	VAR robtarget Openhole_1385 := [[446.82, -4.21, 181.42], [-0.057245, 0.704786, 0.705942, -0.040573], [0,0,0,0], [9E9, 9E9, 9E9, 9E9, 9E9, 9E9]];
	VAR robtarget Openhole_1386 := [[447.31, -4.15, 181.35], [-0.055802, 0.704902, 0.705831, -0.042464], [0,0,0,0], [9E9, 9E9, 9E9, 9E9, 9E9, 9E9]];
	VAR robtarget Openhole_1387 := [[447.8, -4.1, 181.28], [-0.0543, 0.705019, 0.705717, -0.044309], [0,0,0,0], [9E9, 9E9, 9E9, 9E9, 9E9, 9E9]];
	VAR robtarget Openhole_1388 := [[448.3, -4.06, 181.21], [-0.052766, 0.705135, 0.705601, -0.046125], [0,0,0,0], [9E9, 9E9, 9E9, 9E9, 9E9, 9E9]];
	VAR robtarget Openhole_1389 := [[448.79, -4.06, 181.14], [-0.051091, 0.705259, 0.705489, -0.047811], [0,0,0,0], [9E9, 9E9, 9E9, 9E9, 9E9, 9E9]];
	VAR robtarget Openhole_1390 := [[449.78, -4.1, 181], [-0.047615, 0.705502, 0.705261, -0.051054], [0,0,0,0], [9E9, 9E9, 9E9, 9E9, 9E9, 9E9]];
	VAR robtarget Openhole_1391 := [[450.77, -4.2, 180.86], [-0.043933, 0.705741, 0.705037, -0.05406], [0,0,0,0], [9E9, 9E9, 9E9, 9E9, 9E9, 9E9]];
	VAR robtarget Openhole_1392 := [[456.16, -5.01, 180.14], [-0.022875, 0.706737, 0.703678, -0.069553], [0,0,0,0], [9E9, 9E9, 9E9, 9E9, 9E9, 9E9]];
	VAR robtarget Openhole_1393 := [[458.63, -5.19, 179.82], [-0.013826, 0.706972, 0.702881, -0.077186], [0,0,0,0], [9E9, 9E9, 9E9, 9E9, 9E9, 9E9]];
	VAR robtarget Openhole_1394 := [[459.13, -5.2, 179.76], [-0.012101, 0.707003, 0.702703, -0.078798], [0,0,0,0], [9E9, 9E9, 9E9, 9E9, 9E9, 9E9]];
	VAR robtarget Openhole_1395 := [[463.08, -5.04, 179.21], [0.000809, 0.707106, 0.701046, -0.092383], [0,0,0,0], [9E9, 9E9, 9E9, 9E9, 9E9, 9E9]];
	VAR robtarget Openhole_1396 := [[464.07, -4.96, 179.07], [0.003883, 0.707096, 0.700578, -0.095868], [0,0,0,0], [9E9, 9E9, 9E9, 9E9, 9E9, 9E9]];
	VAR robtarget Openhole_1397 := [[472.91, -4.06, 177.66], [0.03065, 0.706442, 0.695628, -0.126894], [0,0,0,0], [9E9, 9E9, 9E9, 9E9, 9E9, 9E9]];
	VAR robtarget Openhole_1398 := [[478.34, -3.86, 176.83], [0.047884, 0.705484, 0.69228, -0.144041], [0,0,0,0], [9E9, 9E9, 9E9, 9E9, 9E9, 9E9]];
	VAR robtarget Openhole_1399 := [[478.84, -3.85, 176.75], [0.049491, 0.705373, 0.691972, -0.145517], [0,0,0,0], [9E9, 9E9, 9E9, 9E9, 9E9, 9E9]];
	VAR robtarget Openhole_1400 := [[479.33, -3.86, 176.68], [0.051109, 0.705257, 0.691664, -0.146975], [0,0,0,0], [9E9, 9E9, 9E9, 9E9, 9E9, 9E9]];
	VAR robtarget Openhole_1401 := [[480.82, -3.88, 176.47], [0.055996, 0.704886, 0.690737, -0.151267], [0,0,0,0], [9E9, 9E9, 9E9, 9E9, 9E9, 9E9]];
	VAR robtarget Openhole_1402 := [[474.12, -5.49, 177.83], [0.039301, 0.706014, 0.69579, -0.126003], [0,0,0,0], [9E9, 9E9, 9E9, 9E9, 9E9, 9E9]];
	VAR robtarget Openhole_1403 := [[469.2, -6.03, 178.58], [0.024725, 0.706674, 0.698676, -0.108864], [0,0,0,0], [9E9, 9E9, 9E9, 9E9, 9E9, 9E9]];
	VAR robtarget Openhole_1404 := [[460.88, -7.27, 179.76], [0.000748, 0.707106, 0.702821, -0.077733], [0,0,0,0], [9E9, 9E9, 9E9, 9E9, 9E9, 9E9]];
	VAR robtarget Openhole_1405 := [[457.42, -7.57, 180.17], [-0.010045, 0.707035, 0.704092, -0.065225], [0,0,0,0], [9E9, 9E9, 9E9, 9E9, 9E9, 9E9]];
	VAR robtarget Openhole_1406 := [[455.43, -7.61, 180.39], [-0.016666, 0.70691, 0.70469, -0.058409], [0,0,0,0], [9E9, 9E9, 9E9, 9E9, 9E9, 9E9]];
	VAR robtarget Openhole_1407 := [[452.45, -7.48, 180.72], [-0.027253, 0.706581, 0.705422, -0.048789], [0,0,0,0], [9E9, 9E9, 9E9, 9E9, 9E9, 9E9]];
	VAR robtarget Openhole_1408 := [[448.48, -7.26, 181.16], [-0.041479, 0.705889, 0.706188, -0.036043], [0,0,0,0], [9E9, 9E9, 9E9, 9E9, 9E9, 9E9]];
	VAR robtarget Openhole_1409 := [[447.49, -7.25, 181.27], [-0.044879, 0.705681, 0.706351, -0.032691], [0,0,0,0], [9E9, 9E9, 9E9, 9E9, 9E9, 9E9]];
	VAR robtarget Openhole_1410 := [[446.49, -7.27, 181.38], [-0.048173, 0.705464, 0.706502, -0.029233], [0,0,0,0], [9E9, 9E9, 9E9, 9E9, 9E9, 9E9]];
	VAR robtarget Openhole_1411 := [[445.5, -7.33, 181.49], [-0.051296, 0.705244, 0.706642, -0.025622], [0,0,0,0], [9E9, 9E9, 9E9, 9E9, 9E9, 9E9]];
	VAR robtarget Openhole_1412 := [[444.51, -7.43, 181.6], [-0.054297, 0.705019, 0.706767, -0.021908], [0,0,0,0], [9E9, 9E9, 9E9, 9E9, 9E9, 9E9]];
	VAR robtarget Openhole_1413 := [[444.02, -7.49, 181.65], [-0.055764, 0.704905, 0.706823, -0.020026], [0,0,0,0], [9E9, 9E9, 9E9, 9E9, 9E9, 9E9]];
	VAR robtarget Openhole_1414 := [[437.6, -8.31, 182.27], [-0.074416, 0.70318, 0.707092, 0.004635], [0,0,0,0], [9E9, 9E9, 9E9, 9E9, 9E9, 9E9]];
	VAR robtarget Openhole_1415 := [[423.69, -9.33, 183.46], [-0.115694, 0.697578, 0.704998, 0.05457], [0,0,0,0], [9E9, 9E9, 9E9, 9E9, 9E9, 9E9]];
	VAR robtarget Openhole_1416 := [[407.25, -10.08, 184.69], [-0.161587, 0.688396, 0.698742, 0.108443], [0,0,0,0], [9E9, 9E9, 9E9, 9E9, 9E9, 9E9]];
	VAR robtarget Openhole_1417 := [[394.36, -10.64, 185.5], [-0.193652, 0.680073, 0.691718, 0.14672], [0,0,0,0], [9E9, 9E9, 9E9, 9E9, 9E9, 9E9]];
	VAR robtarget Openhole_1418 := [[389.36, -10.64, 185.9], [-0.205704, 0.676525, 0.688791, 0.159896], [0,0,0,0], [9E9, 9E9, 9E9, 9E9, 9E9, 9E9]];
	VAR robtarget Openhole_1419 := [[362.36, -10.64, 185.99], [-0.183051, 0.683002, 0.683002, 0.183051], [0,0,0,0], [9E9, 9E9, 9E9, 9E9, 9E9, 9E9]];
	VAR robtarget Openhole_1420 := [[361.72, -33.92, 172.54], [-0.183051, 0.683002, 0.683002, 0.183051], [0,0,0,0], [9E9, 9E9, 9E9, 9E9, 9E9, 9E9]];
	VAR robtarget Openhole_1421 := [[389.32, -33.92, 172.46], [-0.13956, 0.693198, 0.67011, 0.225726], [0,0,0,0], [9E9, 9E9, 9E9, 9E9, 9E9, 9E9]];
	VAR robtarget Openhole_1422 := [[399.12, -33.92, 173.86], [-0.112191, 0.69815, 0.677451, 0.202632], [0,0,0,0], [9E9, 9E9, 9E9, 9E9, 9E9, 9E9]];
	VAR robtarget Openhole_1423 := [[405.5, -35.06, 174.3], [-0.089819, 0.701379, 0.681181, 0.189715], [0,0,0,0], [9E9, 9E9, 9E9, 9E9, 9E9, 9E9]];
	VAR robtarget Openhole_1424 := [[411.91, -35.92, 174.98], [-0.067308, 0.703896, 0.685089, 0.175081], [0,0,0,0], [9E9, 9E9, 9E9, 9E9, 9E9, 9E9]];
	VAR robtarget Openhole_1425 := [[417.83, -36.39, 175.8], [-0.046793, 0.705557, 0.688811, 0.159812], [0,0,0,0], [9E9, 9E9, 9E9, 9E9, 9E9, 9E9]];
	VAR robtarget Openhole_1426 := [[421.78, -36.5, 176.43], [-0.033466, 0.706314, 0.691318, 0.148591], [0,0,0,0], [9E9, 9E9, 9E9, 9E9, 9E9, 9E9]];
	VAR robtarget Openhole_1427 := [[422.28, -36.5, 176.51], [-0.031833, 0.70639, 0.691632, 0.147122], [0,0,0,0], [9E9, 9E9, 9E9, 9E9, 9E9, 9E9]];
	VAR robtarget Openhole_1428 := [[428.18, -36.31, 177.54], [-0.012705, 0.706993, 0.695332, 0.128505], [0,0,0,0], [9E9, 9E9, 9E9, 9E9, 9E9, 9E9]];
	VAR robtarget Openhole_1429 := [[436.05, -35.81, 178.91], [0.012379, 0.706998, 0.699726, 0.101898], [0,0,0,0], [9E9, 9E9, 9E9, 9E9, 9E9, 9E9]];
	VAR robtarget Openhole_1430 := [[437.03, -35.79, 179.08], [0.015677, 0.706933, 0.700196, 0.098619], [0,0,0,0], [9E9, 9E9, 9E9, 9E9, 9E9, 9E9]];
	VAR robtarget Openhole_1431 := [[438.02, -35.8, 179.23], [0.019061, 0.70685, 0.700641, 0.095405], [0,0,0,0], [9E9, 9E9, 9E9, 9E9, 9E9, 9E9]];
	VAR robtarget Openhole_1432 := [[439.01, -35.82, 179.39], [0.022528, 0.706748, 0.701062, 0.092258], [0,0,0,0], [9E9, 9E9, 9E9, 9E9, 9E9, 9E9]];
	VAR robtarget Openhole_1433 := [[439.99, -35.88, 179.55], [0.026095, 0.706625, 0.701458, 0.089204], [0,0,0,0], [9E9, 9E9, 9E9, 9E9, 9E9, 9E9]];
	VAR robtarget Openhole_1434 := [[440.98, -35.98, 179.7], [0.029757, 0.70648, 0.701827, 0.086247], [0,0,0,0], [9E9, 9E9, 9E9, 9E9, 9E9, 9E9]];
	VAR robtarget Openhole_1435 := [[441.96, -36.1, 179.85], [0.03352, 0.706312, 0.702171, 0.083404], [0,0,0,0], [9E9, 9E9, 9E9, 9E9, 9E9, 9E9]];
	VAR robtarget Openhole_1436 := [[442.94, -36.26, 180], [0.037368, 0.706119, 0.702491, 0.080666], [0,0,0,0], [9E9, 9E9, 9E9, 9E9, 9E9, 9E9]];
	VAR robtarget Openhole_1437 := [[443.91, -36.44, 180.15], [0.041287, 0.7059, 0.702789, 0.078026], [0,0,0,0], [9E9, 9E9, 9E9, 9E9, 9E9, 9E9]];
	VAR robtarget Openhole_1438 := [[445.84, -36.87, 180.46], [0.049255, 0.705389, 0.703335, 0.072942], [0,0,0,0], [9E9, 9E9, 9E9, 9E9, 9E9, 9E9]];
	VAR robtarget Openhole_1439 := [[446.31, -37, 180.54], [0.051325, 0.705242, 0.703452, 0.071803], [0,0,0,0], [9E9, 9E9, 9E9, 9E9, 9E9, 9E9]];
	VAR robtarget Openhole_1440 := [[446.78, -37.17, 180.61], [0.05345, 0.705084, 0.703556, 0.070775], [0,0,0,0], [9E9, 9E9, 9E9, 9E9, 9E9, 9E9]];
	VAR robtarget Openhole_1441 := [[447.23, -37.35, 180.69], [0.05561, 0.704917, 0.70365, 0.06983], [0,0,0,0], [9E9, 9E9, 9E9, 9E9, 9E9, 9E9]];
	VAR robtarget Openhole_1442 := [[448.2, -37.57, 180.86], [0.059582, 0.704592, 0.703898, 0.067287], [0,0,0,0], [9E9, 9E9, 9E9, 9E9, 9E9, 9E9]];
	VAR robtarget Openhole_1443 := [[448.69, -37.57, 180.94], [0.061268, 0.704447, 0.704054, 0.06564], [0,0,0,0], [9E9, 9E9, 9E9, 9E9, 9E9, 9E9]];
	VAR robtarget Openhole_1444 := [[449.18, -37.57, 181.03], [0.06291, 0.704303, 0.704209, 0.063947], [0,0,0,0], [9E9, 9E9, 9E9, 9E9, 9E9, 9E9]];
	VAR robtarget Openhole_1445 := [[450.15, -37.36, 181.2], [0.065502, 0.704066, 0.704556, 0.060003], [0,0,0,0], [9E9, 9E9, 9E9, 9E9, 9E9, 9E9]];
	VAR robtarget Openhole_1446 := [[450.62, -37.23, 181.28], [0.066679, 0.703956, 0.704728, 0.057956], [0,0,0,0], [9E9, 9E9, 9E9, 9E9, 9E9, 9E9]];
	VAR robtarget Openhole_1447 := [[451.1, -37.12, 181.37], [0.067916, 0.703838, 0.70489, 0.055943], [0,0,0,0], [9E9, 9E9, 9E9, 9E9, 9E9, 9E9]];
	VAR robtarget Openhole_1448 := [[451.58, -36.98, 181.45], [0.069072, 0.703725, 0.705051, 0.053881], [0,0,0,0], [9E9, 9E9, 9E9, 9E9, 9E9, 9E9]];
	VAR robtarget Openhole_1449 := [[459.65, -34.59, 182.6], [0.088061, 0.701602, 0.706869, 0.01833], [0,0,0,0], [9E9, 9E9, 9E9, 9E9, 9E9, 9E9]];
	VAR robtarget Openhole_1450 := [[460.13, -34.45, 182.66], [0.089197, 0.701458, 0.70692, 0.01625], [0,0,0,0], [9E9, 9E9, 9E9, 9E9, 9E9, 9E9]];
	VAR robtarget Openhole_1451 := [[461.11, -32.96, 182.64], [0.087508, 0.701671, 0.707062, 0.00793], [0,0,0,0], [9E9, 9E9, 9E9, 9E9, 9E9, 9E9]];
	VAR robtarget Openhole_1452 := [[460.14, -33.18, 182.53], [0.085056, 0.701973, 0.707005, 0.01198], [0,0,0,0], [9E9, 9E9, 9E9, 9E9, 9E9, 9E9]];
	VAR robtarget Openhole_1453 := [[453.43, -34.99, 181.69], [0.068762, 0.703755, 0.705919, 0.040973], [0,0,0,0], [9E9, 9E9, 9E9, 9E9, 9E9, 9E9]];
	VAR robtarget Openhole_1454 := [[452.47, -35.23, 181.55], [0.066291, 0.703993, 0.705672, 0.045027], [0,0,0,0], [9E9, 9E9, 9E9, 9E9, 9E9, 9E9]];
	VAR robtarget Openhole_1455 := [[451.98, -35.33, 181.48], [0.065007, 0.704112, 0.705542, 0.047022], [0,0,0,0], [9E9, 9E9, 9E9, 9E9, 9E9, 9E9]];
	VAR robtarget Openhole_1456 := [[451.5, -35.42, 181.4], [0.063682, 0.704233, 0.705408, 0.048988], [0,0,0,0], [9E9, 9E9, 9E9, 9E9, 9E9, 9E9]];
	VAR robtarget Openhole_1457 := [[451.01, -35.49, 181.32], [0.062259, 0.704361, 0.705274, 0.050884], [0,0,0,0], [9E9, 9E9, 9E9, 9E9, 9E9, 9E9]];
	VAR robtarget Openhole_1458 := [[450.52, -35.55, 181.25], [0.06079, 0.704489, 0.705137, 0.052742], [0,0,0,0], [9E9, 9E9, 9E9, 9E9, 9E9, 9E9]];
	VAR robtarget Openhole_1459 := [[450.03, -35.58, 181.17], [0.059241, 0.704621, 0.705001, 0.054535], [0,0,0,0], [9E9, 9E9, 9E9, 9E9, 9E9, 9E9]];
	VAR robtarget Openhole_1460 := [[449.53, -35.6, 181.09], [0.057631, 0.704754, 0.704864, 0.056273], [0,0,0,0], [9E9, 9E9, 9E9, 9E9, 9E9, 9E9]];
	VAR robtarget Openhole_1461 := [[449.04, -35.59, 181.01], [0.055918, 0.704892, 0.704732, 0.057906], [0,0,0,0], [9E9, 9E9, 9E9, 9E9, 9E9, 9E9]];
	VAR robtarget Openhole_1462 := [[448.55, -35.55, 180.93], [0.054128, 0.705032, 0.704603, 0.059455], [0,0,0,0], [9E9, 9E9, 9E9, 9E9, 9E9, 9E9]];
	VAR robtarget Openhole_1463 := [[448.05, -35.5, 180.86], [0.052284, 0.705171, 0.704476, 0.060939], [0,0,0,0], [9E9, 9E9, 9E9, 9E9, 9E9, 9E9]];
	VAR robtarget Openhole_1464 := [[447.57, -35.43, 180.78], [0.050389, 0.705309, 0.704352, 0.062358], [0,0,0,0], [9E9, 9E9, 9E9, 9E9, 9E9, 9E9]];
	VAR robtarget Openhole_1465 := [[446.59, -35.25, 180.63], [0.046491, 0.705577, 0.704108, 0.065048], [0,0,0,0], [9E9, 9E9, 9E9, 9E9, 9E9, 9E9]];
	VAR robtarget Openhole_1466 := [[443.68, -34.65, 180.21], [0.034621, 0.706259, 0.703341, 0.072881], [0,0,0,0], [9E9, 9E9, 9E9, 9E9, 9E9, 9E9]];
	VAR robtarget Openhole_1467 := [[441.72, -34.35, 179.94], [0.026944, 0.706593, 0.702744, 0.078425], [0,0,0,0], [9E9, 9E9, 9E9, 9E9, 9E9, 9E9]];
	VAR robtarget Openhole_1468 := [[440.74, -34.25, 179.8], [0.023237, 0.706725, 0.702411, 0.081357], [0,0,0,0], [9E9, 9E9, 9E9, 9E9, 9E9, 9E9]];
	VAR robtarget Openhole_1469 := [[439.75, -34.17, 179.66], [0.019621, 0.706835, 0.702053, 0.084386], [0,0,0,0], [9E9, 9E9, 9E9, 9E9, 9E9, 9E9]];
	VAR robtarget Openhole_1470 := [[438.76, -34.13, 179.52], [0.016102, 0.706923, 0.701671, 0.087509], [0,0,0,0], [9E9, 9E9, 9E9, 9E9, 9E9, 9E9]];
	VAR robtarget Openhole_1471 := [[437.77, -34.12, 179.38], [0.012688, 0.706993, 0.701262, 0.090726], [0,0,0,0], [9E9, 9E9, 9E9, 9E9, 9E9, 9E9]];
	VAR robtarget Openhole_1472 := [[437.28, -34.12, 179.31], [0.011017, 0.707021, 0.701049, 0.092362], [0,0,0,0], [9E9, 9E9, 9E9, 9E9, 9E9, 9E9]];
	VAR robtarget Openhole_1473 := [[431.85, -34.44, 178.47], [-0.006368, 0.707078, 0.698349, 0.110947], [0,0,0,0], [9E9, 9E9, 9E9, 9E9, 9E9, 9E9]];
	VAR robtarget Openhole_1474 := [[424.96, -34.89, 177.34], [-0.028091, 0.706549, 0.694309, 0.13392], [0,0,0,0], [9E9, 9E9, 9E9, 9E9, 9E9, 9E9]];
	VAR robtarget Openhole_1475 := [[422, -34.94, 176.87], [-0.037745, 0.706099, 0.692485, 0.143054], [0,0,0,0], [9E9, 9E9, 9E9, 9E9, 9E9, 9E9]];
	VAR robtarget Openhole_1476 := [[421.5, -34.94, 176.8], [-0.039386, 0.706009, 0.69218, 0.144521], [0,0,0,0], [9E9, 9E9, 9E9, 9E9, 9E9, 9E9]];
	VAR robtarget Openhole_1477 := [[415.57, -34.71, 175.97], [-0.059446, 0.704604, 0.688505, 0.161124], [0,0,0,0], [9E9, 9E9, 9E9, 9E9, 9E9, 9E9]];
	VAR robtarget Openhole_1478 := [[409.14, -34.09, 175.23], [-0.08164, 0.702378, 0.684557, 0.177147], [0,0,0,0], [9E9, 9E9, 9E9, 9E9, 9E9, 9E9]];
	VAR robtarget Openhole_1479 := [[404.2, -33.45, 174.8], [-0.098663, 0.70019, 0.681563, 0.18834], [0,0,0,0], [9E9, 9E9, 9E9, 9E9, 9E9, 9E9]];
	VAR robtarget Openhole_1480 := [[411.67, -32.92, 176.03], [-0.077413, 0.702856, 0.687197, 0.166612], [0,0,0,0], [9E9, 9E9, 9E9, 9E9, 9E9, 9E9]];
	VAR robtarget Openhole_1481 := [[418.12, -33.28, 176.78], [-0.055758, 0.704905, 0.691162, 0.149313], [0,0,0,0], [9E9, 9E9, 9E9, 9E9, 9E9, 9E9]];
	VAR robtarget Openhole_1482 := [[420.59, -33.32, 177.11], [-0.047583, 0.705504, 0.69268, 0.142107], [0,0,0,0], [9E9, 9E9, 9E9, 9E9, 9E9, 9E9]];
	VAR robtarget Openhole_1483 := [[421.09, -33.31, 177.18], [-0.04597, 0.705611, 0.692983, 0.14062], [0,0,0,0], [9E9, 9E9, 9E9, 9E9, 9E9, 9E9]];
	VAR robtarget Openhole_1484 := [[426.52, -33.08, 177.98], [-0.028736, 0.706523, 0.696271, 0.123317], [0,0,0,0], [9E9, 9E9, 9E9, 9E9, 9E9, 9E9]];
	VAR robtarget Openhole_1485 := [[436.37, -32.09, 179.43], [0.001182, 0.707106, 0.701528, 0.088645], [0,0,0,0], [9E9, 9E9, 9E9, 9E9, 9E9, 9E9]];
	VAR robtarget Openhole_1486 := [[438.84, -31.99, 179.75], [0.009265, 0.707046, 0.702549, 0.080151], [0,0,0,0], [9E9, 9E9, 9E9, 9E9, 9E9, 9E9]];
	VAR robtarget Openhole_1487 := [[439.84, -31.99, 179.88], [0.012667, 0.706993, 0.702914, 0.076885], [0,0,0,0], [9E9, 9E9, 9E9, 9E9, 9E9, 9E9]];
	VAR robtarget Openhole_1488 := [[441.32, -32.04, 180.06], [0.017908, 0.70688, 0.703421, 0.072104], [0,0,0,0], [9E9, 9E9, 9E9, 9E9, 9E9, 9E9]];
	VAR robtarget Openhole_1489 := [[442.32, -32.11, 180.18], [0.0215, 0.70678, 0.703731, 0.069008], [0,0,0,0], [9E9, 9E9, 9E9, 9E9, 9E9, 9E9]];
	VAR robtarget Openhole_1490 := [[442.81, -32.16, 180.24], [0.023347, 0.706721, 0.703876, 0.067516], [0,0,0,0], [9E9, 9E9, 9E9, 9E9, 9E9, 9E9]];
	VAR robtarget Openhole_1491 := [[447.23, -32.82, 180.78], [0.040592, 0.705941, 0.704977, 0.054843], [0,0,0,0], [9E9, 9E9, 9E9, 9E9, 9E9, 9E9]];
	VAR robtarget Openhole_1492 := [[448.21, -32.96, 180.91], [0.044393, 0.705712, 0.705193, 0.051985], [0,0,0,0], [9E9, 9E9, 9E9, 9E9, 9E9, 9E9]];
	VAR robtarget Openhole_1493 := [[448.7, -33.01, 180.97], [0.046239, 0.705593, 0.705302, 0.050486], [0,0,0,0], [9E9, 9E9, 9E9, 9E9, 9E9, 9E9]];
	VAR robtarget Openhole_1494 := [[449.19, -33.05, 181.04], [0.048038, 0.705473, 0.705412, 0.048933], [0,0,0,0], [9E9, 9E9, 9E9, 9E9, 9E9, 9E9]];
	VAR robtarget Openhole_1495 := [[449.69, -33.07, 181.11], [0.049788, 0.705352, 0.705521, 0.047323], [0,0,0,0], [9E9, 9E9, 9E9, 9E9, 9E9, 9E9]];
	VAR robtarget Openhole_1496 := [[450.19, -33.08, 181.17], [0.051486, 0.70523, 0.705631, 0.045656], [0,0,0,0], [9E9, 9E9, 9E9, 9E9, 9E9, 9E9]];
	VAR robtarget Openhole_1497 := [[451.18, -33.03, 181.31], [0.054685, 0.704989, 0.70585, 0.042136], [0,0,0,0], [9E9, 9E9, 9E9, 9E9, 9E9, 9E9]];
	VAR robtarget Openhole_1498 := [[451.67, -32.99, 181.37], [0.056197, 0.70487, 0.705957, 0.0403], [0,0,0,0], [9E9, 9E9, 9E9, 9E9, 9E9, 9E9]];
	VAR robtarget Openhole_1499 := [[452.16, -32.92, 181.44], [0.057637, 0.704754, 0.706063, 0.038404], [0,0,0,0], [9E9, 9E9, 9E9, 9E9, 9E9, 9E9]];
	VAR robtarget Openhole_1500 := [[452.65, -32.84, 181.5], [0.059027, 0.704639, 0.706166, 0.036472], [0,0,0,0], [9E9, 9E9, 9E9, 9E9, 9E9, 9E9]];
	VAR robtarget Openhole_1501 := [[453.62, -32.66, 181.62], [0.061679, 0.704412, 0.706359, 0.032514], [0,0,0,0], [9E9, 9E9, 9E9, 9E9, 9E9, 9E9]];
	VAR robtarget Openhole_1502 := [[460.43, -31.22, 182.36], [0.079553, 0.702618, 0.707093, 0.004412], [0,0,0,0], [9E9, 9E9, 9E9, 9E9, 9E9, 9E9]];
	VAR robtarget Openhole_1503 := [[466.84, -30.31, 182.96], [0.097392, 0.700368, 0.706813, -0.020389], [0,0,0,0], [9E9, 9E9, 9E9, 9E9, 9E9, 9E9]];
	VAR robtarget Openhole_1504 := [[476.26, -29.36, 183.74], [0.123815, 0.696182, 0.704976, -0.054856], [0,0,0,0], [9E9, 9E9, 9E9, 9E9, 9E9, 9E9]];
	VAR robtarget Openhole_1505 := [[470.3, -26.56, 182.58], [0.096146, 0.70054, 0.70571, -0.044425], [0,0,0,0], [9E9, 9E9, 9E9, 9E9, 9E9, 9E9]];
	VAR robtarget Openhole_1506 := [[465.31, -26.64, 182.23], [0.080362, 0.702525, 0.706573, -0.027466], [0,0,0,0], [9E9, 9E9, 9E9, 9E9, 9E9, 9E9]];
	VAR robtarget Openhole_1507 := [[464.81, -26.64, 182.19], [0.078734, 0.70271, 0.706636, -0.02579], [0,0,0,0], [9E9, 9E9, 9E9, 9E9, 9E9, 9E9]];
	VAR robtarget Openhole_1508 := [[463.82, -26.63, 182.12], [0.075461, 0.703069, 0.706751, -0.022436], [0,0,0,0], [9E9, 9E9, 9E9, 9E9, 9E9, 9E9]];
	VAR robtarget Openhole_1509 := [[463.32, -26.64, 182.08], [0.07383, 0.703242, 0.706802, -0.020747], [0,0,0,0], [9E9, 9E9, 9E9, 9E9, 9E9, 9E9]];
	VAR robtarget Openhole_1510 := [[462.82, -26.63, 182.05], [0.072175, 0.703414, 0.706849, -0.019077], [0,0,0,0], [9E9, 9E9, 9E9, 9E9, 9E9, 9E9]];
	VAR robtarget Openhole_1511 := [[459.33, -26.59, 181.79], [0.060506, 0.704513, 0.707069, -0.007354], [0,0,0,0], [9E9, 9E9, 9E9, 9E9, 9E9, 9E9]];
	VAR robtarget Openhole_1512 := [[458.83, -26.59, 181.75], [0.058846, 0.704654, 0.707084, -0.005656], [0,0,0,0], [9E9, 9E9, 9E9, 9E9, 9E9, 9E9]];
	VAR robtarget Openhole_1513 := [[458.33, -26.6, 181.72], [0.057195, 0.70479, 0.707096, -0.003946], [0,0,0,0], [9E9, 9E9, 9E9, 9E9, 9E9, 9E9]];
	VAR robtarget Openhole_1514 := [[457.83, -26.59, 181.68], [0.055521, 0.704924, 0.707103, -0.002257], [0,0,0,0], [9E9, 9E9, 9E9, 9E9, 9E9, 9E9]];
	VAR robtarget Openhole_1515 := [[456.34, -26.58, 181.57], [0.050456, 0.705304, 0.707101, 0.002786], [0,0,0,0], [9E9, 9E9, 9E9, 9E9, 9E9, 9E9]];
	VAR robtarget Openhole_1516 := [[455.34, -26.54, 181.49], [0.046991, 0.705544, 0.707081, 0.006067], [0,0,0,0], [9E9, 9E9, 9E9, 9E9, 9E9, 9E9]];
	VAR robtarget Openhole_1517 := [[454.84, -26.49, 181.46], [0.045165, 0.705663, 0.707066, 0.007603], [0,0,0,0], [9E9, 9E9, 9E9, 9E9, 9E9, 9E9]];
	VAR robtarget Openhole_1518 := [[454.35, -26.44, 181.42], [0.043303, 0.70578, 0.707048, 0.009097], [0,0,0,0], [9E9, 9E9, 9E9, 9E9, 9E9, 9E9]];
	VAR robtarget Openhole_1519 := [[453.86, -26.35, 181.38], [0.041367, 0.705896, 0.707029, 0.010494], [0,0,0,0], [9E9, 9E9, 9E9, 9E9, 9E9, 9E9]];
	VAR robtarget Openhole_1520 := [[453.37, -26.25, 181.34], [0.039385, 0.706009, 0.707008, 0.011826], [0,0,0,0], [9E9, 9E9, 9E9, 9E9, 9E9, 9E9]];
	VAR robtarget Openhole_1521 := [[452.79, -25.92, 181.29], [0.0363, 0.706174, 0.706993, 0.012685], [0,0,0,0], [9E9, 9E9, 9E9, 9E9, 9E9, 9E9]];
	VAR robtarget Openhole_1522 := [[454.94, -24.42, 181.35], [0.038494, 0.706058, 0.707107, 0.000235], [0,0,0,0], [9E9, 9E9, 9E9, 9E9, 9E9, 9E9]];
	VAR robtarget Openhole_1523 := [[455.54, -24.57, 181.39], [0.041032, 0.705915, 0.707106, -0.001297], [0,0,0,0], [9E9, 9E9, 9E9, 9E9, 9E9, 9E9]];
	VAR robtarget Openhole_1524 := [[456.54, -24.66, 181.45], [0.044665, 0.705695, 0.707093, -0.004397], [0,0,0,0], [9E9, 9E9, 9E9, 9E9, 9E9, 9E9]];
	VAR robtarget Openhole_1525 := [[457.04, -24.68, 181.48], [0.046428, 0.705581, 0.707081, -0.006004], [0,0,0,0], [9E9, 9E9, 9E9, 9E9, 9E9, 9E9]];
	VAR robtarget Openhole_1526 := [[460.52, -24.98, 181.7], [0.059039, 0.704638, 0.706906, -0.016839], [0,0,0,0], [9E9, 9E9, 9E9, 9E9, 9E9, 9E9]];
	VAR robtarget Openhole_1527 := [[457.18, -28.45, 181.77], [0.059563, 0.704594, 0.707079, 0.006212], [0,0,0,0], [9E9, 9E9, 9E9, 9E9, 9E9, 9E9]];
	VAR robtarget Openhole_1528 := [[454.2, -28.65, 181.51], [0.050244, 0.705319, 0.706901, 0.017075], [0,0,0,0], [9E9, 9E9, 9E9, 9E9, 9E9, 9E9]];
	VAR robtarget Openhole_1529 := [[453.7, -28.66, 181.47], [0.048609, 0.705434, 0.706856, 0.018817], [0,0,0,0], [9E9, 9E9, 9E9, 9E9, 9E9, 9E9]];
	VAR robtarget Openhole_1530 := [[452.71, -28.67, 181.37], [0.045277, 0.705656, 0.706757, 0.022241], [0,0,0,0], [9E9, 9E9, 9E9, 9E9, 9E9, 9E9]];
	VAR robtarget Openhole_1531 := [[449.23, -28.52, 181.05], [0.033008, 0.706336, 0.706307, 0.033626], [0,0,0,0], [9E9, 9E9, 9E9, 9E9, 9E9, 9E9]];
	VAR robtarget Openhole_1532 := [[448.73, -28.52, 181.01], [0.031293, 0.706414, 0.706225, 0.035294], [0,0,0,0], [9E9, 9E9, 9E9, 9E9, 9E9, 9E9]];
	VAR robtarget Openhole_1533 := [[448.23, -28.52, 180.96], [0.029603, 0.706487, 0.706139, 0.036988], [0,0,0,0], [9E9, 9E9, 9E9, 9E9, 9E9, 9E9]];
	VAR robtarget Openhole_1534 := [[447.24, -28.52, 180.87], [0.02623, 0.70662, 0.705953, 0.040382], [0,0,0,0], [9E9, 9E9, 9E9, 9E9, 9E9, 9E9]];
	VAR robtarget Openhole_1535 := [[444.75, -28.61, 180.64], [0.018061, 0.706876, 0.7054, 0.049099], [0,0,0,0], [9E9, 9E9, 9E9, 9E9, 9E9, 9E9]];
	VAR robtarget Openhole_1536 := [[443.26, -28.67, 180.5], [0.013204, 0.706983, 0.705015, 0.054352], [0,0,0,0], [9E9, 9E9, 9E9, 9E9, 9E9, 9E9]];
	VAR robtarget Openhole_1537 := [[444.55, -31.6, 180.48], [0.027447, 0.706574, 0.704572, 0.059817], [0,0,0,0], [9E9, 9E9, 9E9, 9E9, 9E9, 9E9]];
	VAR robtarget Openhole_1538 := [[445.54, -31.73, 180.6], [0.03123, 0.706417, 0.704812, 0.056924], [0,0,0,0], [9E9, 9E9, 9E9, 9E9, 9E9, 9E9]];
	VAR robtarget Openhole_1539 := [[446.52, -31.9, 180.71], [0.035109, 0.706235, 0.70503, 0.05416], [0,0,0,0], [9E9, 9E9, 9E9, 9E9, 9E9, 9E9]];
	VAR robtarget Openhole_1540 := [[448.49, -32.14, 180.95], [0.042616, 0.705821, 0.705455, 0.048298], [0,0,0,0], [9E9, 9E9, 9E9, 9E9, 9E9, 9E9]];
	VAR robtarget Openhole_1541 := [[448.98, -32.18, 181.02], [0.044435, 0.705709, 0.705559, 0.046761], [0,0,0,0], [9E9, 9E9, 9E9, 9E9, 9E9, 9E9]];
	VAR robtarget Openhole_1542 := [[449.48, -32.21, 181.08], [0.046209, 0.705595, 0.705662, 0.045173], [0,0,0,0], [9E9, 9E9, 9E9, 9E9, 9E9, 9E9]];
	VAR robtarget Openhole_1543 := [[449.97, -32.23, 181.14], [0.047949, 0.705479, 0.705764, 0.043549], [0,0,0,0], [9E9, 9E9, 9E9, 9E9, 9E9, 9E9]];
	VAR robtarget Openhole_1544 := [[450.47, -32.23, 181.2], [0.049624, 0.705363, 0.705867, 0.041855], [0,0,0,0], [9E9, 9E9, 9E9, 9E9, 9E9, 9E9]];
	VAR robtarget Openhole_1545 := [[450.96, -32.22, 181.27], [0.051253, 0.705247, 0.705968, 0.04012], [0,0,0,0], [9E9, 9E9, 9E9, 9E9, 9E9, 9E9]];
	VAR robtarget Openhole_1546 := [[451.46, -32.18, 181.33], [0.052812, 0.705132, 0.706068, 0.038318], [0,0,0,0], [9E9, 9E9, 9E9, 9E9, 9E9, 9E9]];
	VAR robtarget Openhole_1547 := [[451.95, -32.13, 181.39], [0.05432, 0.705017, 0.706165, 0.036474], [0,0,0,0], [9E9, 9E9, 9E9, 9E9, 9E9, 9E9]];
	VAR robtarget Openhole_1548 := [[452.45, -32.07, 181.45], [0.055766, 0.704904, 0.706261, 0.03458], [0,0,0,0], [9E9, 9E9, 9E9, 9E9, 9E9, 9E9]];
	VAR robtarget Openhole_1549 := [[453.43, -31.9, 181.57], [0.058505, 0.704682, 0.706441, 0.030677], [0,0,0,0], [9E9, 9E9, 9E9, 9E9, 9E9, 9E9]];
	VAR robtarget Openhole_1550 := [[452.74, -30.49, 181.44], [0.051498, 0.705229, 0.706541, 0.028284], [0,0,0,0], [9E9, 9E9, 9E9, 9E9, 9E9, 9E9]];
	VAR robtarget Openhole_1551 := [[451.25, -30.57, 181.27], [0.046727, 0.705561, 0.706307, 0.033621], [0,0,0,0], [9E9, 9E9, 9E9, 9E9, 9E9, 9E9]];
	VAR robtarget Openhole_1552 := [[450.75, -30.57, 181.22], [0.045054, 0.70567, 0.706224, 0.035323], [0,0,0,0], [9E9, 9E9, 9E9, 9E9, 9E9, 9E9]];
	VAR robtarget Openhole_1553 := [[450.26, -30.57, 181.16], [0.043355, 0.705776, 0.706138, 0.036998], [0,0,0,0], [9E9, 9E9, 9E9, 9E9, 9E9, 9E9]];
	VAR robtarget Openhole_1554 := [[446.79, -30.31, 180.78], [0.030739, 0.706438, 0.70548, 0.047944], [0,0,0,0], [9E9, 9E9, 9E9, 9E9, 9E9, 9E9]];
	VAR robtarget Openhole_1555 := [[446.79, -30.31, 180.9], [0.030776, 0.706437, 0.705483, 0.047888], [0,0,0,0], [9E9, 9E9, 9E9, 9E9, 9E9, 9E9]];
	VAR robtarget Openhole_1556 := [[450.26, -30.57, 181.28], [0.043406, 0.705773, 0.70614, 0.036954], [0,0,0,0], [9E9, 9E9, 9E9, 9E9, 9E9, 9E9]];
	VAR robtarget Openhole_1557 := [[450.75, -30.57, 181.34], [0.045107, 0.705667, 0.706226, 0.035281], [0,0,0,0], [9E9, 9E9, 9E9, 9E9, 9E9, 9E9]];
	VAR robtarget Openhole_1558 := [[451.25, -30.57, 181.39], [0.046782, 0.705558, 0.706309, 0.033581], [0,0,0,0], [9E9, 9E9, 9E9, 9E9, 9E9, 9E9]];
	VAR robtarget Openhole_1559 := [[452.74, -30.49, 181.56], [0.051558, 0.705225, 0.706542, 0.02825], [0,0,0,0], [9E9, 9E9, 9E9, 9E9, 9E9, 9E9]];
	VAR robtarget Openhole_1560 := [[453.43, -31.9, 181.69], [0.058572, 0.704677, 0.706443, 0.03064], [0,0,0,0], [9E9, 9E9, 9E9, 9E9, 9E9, 9E9]];
	VAR robtarget Openhole_1561 := [[452.45, -32.07, 181.57], [0.055831, 0.704899, 0.706263, 0.034539], [0,0,0,0], [9E9, 9E9, 9E9, 9E9, 9E9, 9E9]];
	VAR robtarget Openhole_1562 := [[451.95, -32.13, 181.51], [0.054383, 0.705012, 0.706168, 0.036431], [0,0,0,0], [9E9, 9E9, 9E9, 9E9, 9E9, 9E9]];
	VAR robtarget Openhole_1563 := [[451.46, -32.18, 181.45], [0.052873, 0.705127, 0.70607, 0.038273], [0,0,0,0], [9E9, 9E9, 9E9, 9E9, 9E9, 9E9]];
	VAR robtarget Openhole_1564 := [[450.97, -32.22, 181.39], [0.051313, 0.705243, 0.70597, 0.040073], [0,0,0,0], [9E9, 9E9, 9E9, 9E9, 9E9, 9E9]];
	VAR robtarget Openhole_1565 := [[450.47, -32.23, 181.32], [0.049681, 0.705359, 0.70587, 0.041806], [0,0,0,0], [9E9, 9E9, 9E9, 9E9, 9E9, 9E9]];
	VAR robtarget Openhole_1566 := [[449.97, -32.23, 181.26], [0.048005, 0.705475, 0.705768, 0.043498], [0,0,0,0], [9E9, 9E9, 9E9, 9E9, 9E9, 9E9]];
	VAR robtarget Openhole_1567 := [[449.48, -32.21, 181.2], [0.046263, 0.705592, 0.705666, 0.04512], [0,0,0,0], [9E9, 9E9, 9E9, 9E9, 9E9, 9E9]];
	VAR robtarget Openhole_1568 := [[448.98, -32.18, 181.14], [0.044487, 0.705706, 0.705563, 0.046706], [0,0,0,0], [9E9, 9E9, 9E9, 9E9, 9E9, 9E9]];
	VAR robtarget Openhole_1569 := [[448.49, -32.14, 181.07], [0.042666, 0.705818, 0.705459, 0.048242], [0,0,0,0], [9E9, 9E9, 9E9, 9E9, 9E9, 9E9]];
	VAR robtarget Openhole_1570 := [[446.52, -31.9, 180.83], [0.035151, 0.706233, 0.705034, 0.054097], [0,0,0,0], [9E9, 9E9, 9E9, 9E9, 9E9, 9E9]];
	VAR robtarget Openhole_1571 := [[445.54, -31.73, 180.72], [0.031267, 0.706415, 0.704817, 0.056859], [0,0,0,0], [9E9, 9E9, 9E9, 9E9, 9E9, 9E9]];
	VAR robtarget Openhole_1572 := [[444.55, -31.6, 180.6], [0.02748, 0.706573, 0.704578, 0.059749], [0,0,0,0], [9E9, 9E9, 9E9, 9E9, 9E9, 9E9]];
	VAR robtarget Openhole_1573 := [[443.26, -28.67, 180.62], [0.013221, 0.706983, 0.70502, 0.054289], [0,0,0,0], [9E9, 9E9, 9E9, 9E9, 9E9, 9E9]];
	VAR robtarget Openhole_1574 := [[444.75, -28.61, 180.76], [0.018083, 0.706876, 0.705404, 0.049042], [0,0,0,0], [9E9, 9E9, 9E9, 9E9, 9E9, 9E9]];
	VAR robtarget Openhole_1575 := [[447.24, -28.52, 180.99], [0.026262, 0.706619, 0.705955, 0.040334], [0,0,0,0], [9E9, 9E9, 9E9, 9E9, 9E9, 9E9]];
	VAR robtarget Openhole_1576 := [[448.73, -28.52, 181.13], [0.03133, 0.706412, 0.706228, 0.035252], [0,0,0,0], [9E9, 9E9, 9E9, 9E9, 9E9, 9E9]];
	VAR robtarget Openhole_1577 := [[449.23, -28.52, 181.17], [0.033047, 0.706334, 0.706309, 0.033586], [0,0,0,0], [9E9, 9E9, 9E9, 9E9, 9E9, 9E9]];
	VAR robtarget Openhole_1578 := [[452.71, -28.67, 181.49], [0.045329, 0.705652, 0.706758, 0.022214], [0,0,0,0], [9E9, 9E9, 9E9, 9E9, 9E9, 9E9]];
	VAR robtarget Openhole_1579 := [[453.71, -28.66, 181.59], [0.048666, 0.70543, 0.706857, 0.018793], [0,0,0,0], [9E9, 9E9, 9E9, 9E9, 9E9, 9E9]];
	VAR robtarget Openhole_1580 := [[454.2, -28.65, 181.63], [0.050303, 0.705315, 0.706901, 0.017054], [0,0,0,0], [9E9, 9E9, 9E9, 9E9, 9E9, 9E9]];
	VAR robtarget Openhole_1581 := [[457.18, -28.45, 181.89], [0.059632, 0.704588, 0.70708, 0.006203], [0,0,0,0], [9E9, 9E9, 9E9, 9E9, 9E9, 9E9]];
	VAR robtarget Openhole_1582 := [[460.52, -24.98, 181.82], [0.059107, 0.704632, 0.706907, -0.016821], [0,0,0,0], [9E9, 9E9, 9E9, 9E9, 9E9, 9E9]];
	VAR robtarget Openhole_1583 := [[457.04, -24.68, 181.6], [0.046482, 0.705577, 0.707081, -0.005999], [0,0,0,0], [9E9, 9E9, 9E9, 9E9, 9E9, 9E9]];
	VAR robtarget Openhole_1584 := [[456.54, -24.66, 181.57], [0.044717, 0.705691, 0.707093, -0.004393], [0,0,0,0], [9E9, 9E9, 9E9, 9E9, 9E9, 9E9]];
	VAR robtarget Openhole_1585 := [[455.54, -24.57, 181.51], [0.04108, 0.705912, 0.707106, -0.001297], [0,0,0,0], [9E9, 9E9, 9E9, 9E9, 9E9, 9E9]];
	VAR robtarget Openhole_1586 := [[454.94, -24.42, 181.47], [0.03854, 0.706056, 0.707107, 0.000233], [0,0,0,0], [9E9, 9E9, 9E9, 9E9, 9E9, 9E9]];
	VAR robtarget Openhole_1587 := [[452.79, -25.92, 181.41], [0.036343, 0.706172, 0.706993, 0.012669], [0,0,0,0], [9E9, 9E9, 9E9, 9E9, 9E9, 9E9]];
	VAR robtarget Openhole_1588 := [[453.37, -26.25, 181.46], [0.039431, 0.706007, 0.707008, 0.011811], [0,0,0,0], [9E9, 9E9, 9E9, 9E9, 9E9, 9E9]];
	VAR robtarget Openhole_1589 := [[453.86, -26.35, 181.5], [0.041416, 0.705893, 0.707029, 0.01048], [0,0,0,0], [9E9, 9E9, 9E9, 9E9, 9E9, 9E9]];
	VAR robtarget Openhole_1590 := [[454.35, -26.44, 181.54], [0.043354, 0.705776, 0.707048, 0.009085], [0,0,0,0], [9E9, 9E9, 9E9, 9E9, 9E9, 9E9]];
	VAR robtarget Openhole_1591 := [[454.84, -26.49, 181.58], [0.045218, 0.70566, 0.707066, 0.007592], [0,0,0,0], [9E9, 9E9, 9E9, 9E9, 9E9, 9E9]];
	VAR robtarget Openhole_1592 := [[455.34, -26.54, 181.61], [0.047046, 0.70554, 0.707081, 0.006058], [0,0,0,0], [9E9, 9E9, 9E9, 9E9, 9E9, 9E9]];
	VAR robtarget Openhole_1593 := [[456.34, -26.58, 181.69], [0.050515, 0.7053, 0.707101, 0.002781], [0,0,0,0], [9E9, 9E9, 9E9, 9E9, 9E9, 9E9]];
	VAR robtarget Openhole_1594 := [[458.33, -26.6, 181.84], [0.057261, 0.704785, 0.707096, -0.003943], [0,0,0,0], [9E9, 9E9, 9E9, 9E9, 9E9, 9E9]];
	VAR robtarget Openhole_1595 := [[458.83, -26.59, 181.87], [0.058914, 0.704648, 0.707084, -0.005651], [0,0,0,0], [9E9, 9E9, 9E9, 9E9, 9E9, 9E9]];
	VAR robtarget Openhole_1596 := [[459.33, -26.59, 181.91], [0.060575, 0.704507, 0.707069, -0.007347], [0,0,0,0], [9E9, 9E9, 9E9, 9E9, 9E9, 9E9]];
	VAR robtarget Openhole_1597 := [[459.83, -26.6, 181.95], [0.062246, 0.704362, 0.707049, -0.00903], [0,0,0,0], [9E9, 9E9, 9E9, 9E9, 9E9, 9E9]];
	VAR robtarget Openhole_1598 := [[463.32, -26.64, 182.2], [0.073913, 0.703233, 0.706803, -0.020725], [0,0,0,0], [9E9, 9E9, 9E9, 9E9, 9E9, 9E9]];
	VAR robtarget Openhole_1599 := [[463.82, -26.63, 182.24], [0.075546, 0.70306, 0.706751, -0.022413], [0,0,0,0], [9E9, 9E9, 9E9, 9E9, 9E9, 9E9]];
	VAR robtarget Openhole_1600 := [[464.32, -26.64, 182.28], [0.077188, 0.702881, 0.706696, -0.024087], [0,0,0,0], [9E9, 9E9, 9E9, 9E9, 9E9, 9E9]];
	VAR robtarget Openhole_1601 := [[465.31, -26.64, 182.35], [0.080452, 0.702515, 0.706574, -0.027437], [0,0,0,0], [9E9, 9E9, 9E9, 9E9, 9E9, 9E9]];
	VAR robtarget Openhole_1602 := [[465.81, -26.64, 182.39], [0.082068, 0.702328, 0.706507, -0.029121], [0,0,0,0], [9E9, 9E9, 9E9, 9E9, 9E9, 9E9]];
	VAR robtarget Openhole_1603 := [[470.3, -26.56, 182.7], [0.09625, 0.700525, 0.705713, -0.044378], [0,0,0,0], [9E9, 9E9, 9E9, 9E9, 9E9, 9E9]];
	VAR robtarget Openhole_1604 := [[476.26, -29.36, 183.86], [0.123944, 0.696159, 0.70498, -0.054801], [0,0,0,0], [9E9, 9E9, 9E9, 9E9, 9E9, 9E9]];
	VAR robtarget Openhole_1605 := [[466.35, -30.36, 183.04], [0.096097, 0.700547, 0.706865, -0.018508], [0,0,0,0], [9E9, 9E9, 9E9, 9E9, 9E9, 9E9]];
	VAR robtarget Openhole_1606 := [[460.43, -31.22, 182.48], [0.079642, 0.702607, 0.707093, 0.004405], [0,0,0,0], [9E9, 9E9, 9E9, 9E9, 9E9, 9E9]];
	VAR robtarget Openhole_1607 := [[453.63, -32.66, 181.74], [0.061749, 0.704405, 0.706361, 0.032475], [0,0,0,0], [9E9, 9E9, 9E9, 9E9, 9E9, 9E9]];
	VAR robtarget Openhole_1608 := [[452.65, -32.84, 181.62], [0.059095, 0.704633, 0.706168, 0.036428], [0,0,0,0], [9E9, 9E9, 9E9, 9E9, 9E9, 9E9]];
	VAR robtarget Openhole_1609 := [[452.16, -32.92, 181.56], [0.057703, 0.704748, 0.706066, 0.038359], [0,0,0,0], [9E9, 9E9, 9E9, 9E9, 9E9, 9E9]];
	VAR robtarget Openhole_1610 := [[451.67, -32.99, 181.49], [0.056262, 0.704865, 0.70596, 0.040252], [0,0,0,0], [9E9, 9E9, 9E9, 9E9, 9E9, 9E9]];
	VAR robtarget Openhole_1611 := [[451.18, -33.03, 181.43], [0.054748, 0.704984, 0.705853, 0.042086], [0,0,0,0], [9E9, 9E9, 9E9, 9E9, 9E9, 9E9]];
	VAR robtarget Openhole_1612 := [[450.19, -33.08, 181.29], [0.051546, 0.705226, 0.705635, 0.045602], [0,0,0,0], [9E9, 9E9, 9E9, 9E9, 9E9, 9E9]];
	VAR robtarget Openhole_1613 := [[449.69, -33.07, 181.23], [0.049846, 0.705348, 0.705525, 0.047267], [0,0,0,0], [9E9, 9E9, 9E9, 9E9, 9E9, 9E9]];
	VAR robtarget Openhole_1614 := [[449.19, -33.05, 181.16], [0.048094, 0.705469, 0.705416, 0.048876], [0,0,0,0], [9E9, 9E9, 9E9, 9E9, 9E9, 9E9]];
	VAR robtarget Openhole_1615 := [[448.7, -33.01, 181.09], [0.046293, 0.70559, 0.705306, 0.050428], [0,0,0,0], [9E9, 9E9, 9E9, 9E9, 9E9, 9E9]];
	VAR robtarget Openhole_1616 := [[448.21, -32.96, 181.03], [0.044445, 0.705709, 0.705198, 0.051925], [0,0,0,0], [9E9, 9E9, 9E9, 9E9, 9E9, 9E9]];
	VAR robtarget Openhole_1617 := [[447.23, -32.82, 180.9], [0.040639, 0.705938, 0.704982, 0.05478], [0,0,0,0], [9E9, 9E9, 9E9, 9E9, 9E9, 9E9]];
	VAR robtarget Openhole_1618 := [[442.81, -32.16, 180.36], [0.023375, 0.70672, 0.703883, 0.067439], [0,0,0,0], [9E9, 9E9, 9E9, 9E9, 9E9, 9E9]];
	VAR robtarget Openhole_1619 := [[442.32, -32.11, 180.3], [0.021526, 0.706779, 0.703739, 0.06893], [0,0,0,0], [9E9, 9E9, 9E9, 9E9, 9E9, 9E9]];
	VAR robtarget Openhole_1620 := [[441.32, -32.04, 180.18], [0.017931, 0.706879, 0.703429, 0.072022], [0,0,0,0], [9E9, 9E9, 9E9, 9E9, 9E9, 9E9]];
	VAR robtarget Openhole_1621 := [[439.84, -31.99, 180], [0.012684, 0.706993, 0.702924, 0.076798], [0,0,0,0], [9E9, 9E9, 9E9, 9E9, 9E9, 9E9]];
	VAR robtarget Openhole_1622 := [[438.84, -31.99, 179.87], [0.009278, 0.707046, 0.70256, 0.080061], [0,0,0,0], [9E9, 9E9, 9E9, 9E9, 9E9, 9E9]];
	VAR robtarget Openhole_1623 := [[434.39, -32.25, 179.28], [-0.004974, 0.707089, 0.700625, 0.095521], [0,0,0,0], [9E9, 9E9, 9E9, 9E9, 9E9, 9E9]];
	VAR robtarget Openhole_1624 := [[426.03, -33.12, 178.02], [-0.030285, 0.706458, 0.696, 0.124837], [0,0,0,0], [9E9, 9E9, 9E9, 9E9, 9E9, 9E9]];
	VAR robtarget Openhole_1625 := [[420.59, -33.32, 177.23], [-0.047629, 0.705501, 0.692709, 0.141964], [0,0,0,0], [9E9, 9E9, 9E9, 9E9, 9E9, 9E9]];
	VAR robtarget Openhole_1626 := [[420.1, -33.31, 177.16], [-0.049254, 0.705389, 0.692407, 0.143432], [0,0,0,0], [9E9, 9E9, 9E9, 9E9, 9E9, 9E9]];
	VAR robtarget Openhole_1627 := [[413.65, -33.07, 176.36], [-0.070773, 0.703556, 0.688452, 0.16135], [0,0,0,0], [9E9, 9E9, 9E9, 9E9, 9E9, 9E9]];
	VAR robtarget Openhole_1628 := [[411.67, -32.92, 176.15], [-0.077486, 0.702848, 0.687235, 0.166456], [0,0,0,0], [9E9, 9E9, 9E9, 9E9, 9E9, 9E9]];
	VAR robtarget Openhole_1629 := [[404.2, -33.45, 174.92], [-0.09875, 0.700177, 0.681609, 0.188175], [0,0,0,0], [9E9, 9E9, 9E9, 9E9, 9E9, 9E9]];
	VAR robtarget Openhole_1630 := [[411.12, -34.32, 175.56], [-0.07486, 0.703133, 0.685805, 0.172256], [0,0,0,0], [9E9, 9E9, 9E9, 9E9, 9E9, 9E9]];
	VAR robtarget Openhole_1631 := [[417.05, -34.8, 176.28], [-0.05442, 0.70501, 0.689457, 0.156999], [0,0,0,0], [9E9, 9E9, 9E9, 9E9, 9E9, 9E9]];
	VAR robtarget Openhole_1632 := [[422, -34.94, 176.99], [-0.03778, 0.706097, 0.692515, 0.142911], [0,0,0,0], [9E9, 9E9, 9E9, 9E9, 9E9, 9E9]];
	VAR robtarget Openhole_1633 := [[422.49, -34.94, 177.07], [-0.036154, 0.706182, 0.69282, 0.141421], [0,0,0,0], [9E9, 9E9, 9E9, 9E9, 9E9, 9E9]];
	VAR robtarget Openhole_1634 := [[428.41, -34.71, 178.02], [-0.017144, 0.706899, 0.696407, 0.122547], [0,0,0,0], [9E9, 9E9, 9E9, 9E9, 9E9, 9E9]];
	VAR robtarget Openhole_1635 := [[436.29, -34.15, 179.28], [0.007744, 0.707064, 0.700618, 0.095572], [0,0,0,0], [9E9, 9E9, 9E9, 9E9, 9E9, 9E9]];
	VAR robtarget Openhole_1636 := [[437.77, -34.12, 179.5], [0.012706, 0.706993, 0.701275, 0.090626], [0,0,0,0], [9E9, 9E9, 9E9, 9E9, 9E9, 9E9]];
	VAR robtarget Openhole_1637 := [[438.27, -34.12, 179.57], [0.014404, 0.70696, 0.701482, 0.08901], [0,0,0,0], [9E9, 9E9, 9E9, 9E9, 9E9, 9E9]];
	VAR robtarget Openhole_1638 := [[438.76, -34.13, 179.64], [0.016123, 0.706923, 0.701683, 0.087412], [0,0,0,0], [9E9, 9E9, 9E9, 9E9, 9E9, 9E9]];
	VAR robtarget Openhole_1639 := [[439.75, -34.17, 179.78], [0.019646, 0.706834, 0.702065, 0.084292], [0,0,0,0], [9E9, 9E9, 9E9, 9E9, 9E9, 9E9]];
	VAR robtarget Openhole_1640 := [[440.74, -34.25, 179.92], [0.023266, 0.706724, 0.702421, 0.081266], [0,0,0,0], [9E9, 9E9, 9E9, 9E9, 9E9, 9E9]];
	VAR robtarget Openhole_1641 := [[441.72, -34.35, 180.06], [0.026977, 0.706592, 0.702754, 0.078337], [0,0,0,0], [9E9, 9E9, 9E9, 9E9, 9E9, 9E9]];
	VAR robtarget Openhole_1642 := [[443.68, -34.65, 180.33], [0.034663, 0.706257, 0.703349, 0.072798], [0,0,0,0], [9E9, 9E9, 9E9, 9E9, 9E9, 9E9]];
	VAR robtarget Openhole_1643 := [[446.59, -35.25, 180.75], [0.046545, 0.705573, 0.704115, 0.064974], [0,0,0,0], [9E9, 9E9, 9E9, 9E9, 9E9, 9E9]];
	VAR robtarget Openhole_1644 := [[447.57, -35.43, 180.9], [0.050448, 0.705305, 0.704358, 0.062287], [0,0,0,0], [9E9, 9E9, 9E9, 9E9, 9E9, 9E9]];
	VAR robtarget Openhole_1645 := [[448.05, -35.5, 180.98], [0.052344, 0.705167, 0.704482, 0.060869], [0,0,0,0], [9E9, 9E9, 9E9, 9E9, 9E9, 9E9]];
	VAR robtarget Openhole_1646 := [[448.55, -35.55, 181.05], [0.054191, 0.705027, 0.704609, 0.059386], [0,0,0,0], [9E9, 9E9, 9E9, 9E9, 9E9, 9E9]];
	VAR robtarget Openhole_1647 := [[449.04, -35.59, 181.13], [0.055983, 0.704887, 0.704737, 0.05784], [0,0,0,0], [9E9, 9E9, 9E9, 9E9, 9E9, 9E9]];
	VAR robtarget Openhole_1648 := [[449.53, -35.6, 181.21], [0.057697, 0.704749, 0.704869, 0.056207], [0,0,0,0], [9E9, 9E9, 9E9, 9E9, 9E9, 9E9]];
	VAR robtarget Openhole_1649 := [[450.03, -35.58, 181.29], [0.059309, 0.704615, 0.705006, 0.054472], [0,0,0,0], [9E9, 9E9, 9E9, 9E9, 9E9, 9E9]];
	VAR robtarget Openhole_1650 := [[450.52, -35.55, 181.37], [0.060859, 0.704483, 0.705142, 0.052681], [0,0,0,0], [9E9, 9E9, 9E9, 9E9, 9E9, 9E9]];
	VAR robtarget Openhole_1651 := [[451.01, -35.49, 181.44], [0.06233, 0.704354, 0.705278, 0.050825], [0,0,0,0], [9E9, 9E9, 9E9, 9E9, 9E9, 9E9]];
	VAR robtarget Openhole_1652 := [[451.5, -35.42, 181.52], [0.063755, 0.704227, 0.705412, 0.048931], [0,0,0,0], [9E9, 9E9, 9E9, 9E9, 9E9, 9E9]];
	VAR robtarget Openhole_1653 := [[451.98, -35.33, 181.6], [0.065081, 0.704105, 0.705545, 0.046967], [0,0,0,0], [9E9, 9E9, 9E9, 9E9, 9E9, 9E9]];
	VAR robtarget Openhole_1654 := [[452.47, -35.23, 181.67], [0.066366, 0.703985, 0.705675, 0.044974], [0,0,0,0], [9E9, 9E9, 9E9, 9E9, 9E9, 9E9]];
	VAR robtarget Openhole_1655 := [[453.43, -34.99, 181.81], [0.06884, 0.703748, 0.705922, 0.040924], [0,0,0,0], [9E9, 9E9, 9E9, 9E9, 9E9, 9E9]];
	VAR robtarget Openhole_1656 := [[460.14, -33.18, 182.65], [0.085151, 0.701961, 0.707006, 0.011964], [0,0,0,0], [9E9, 9E9, 9E9, 9E9, 9E9, 9E9]];
	VAR robtarget Openhole_1657 := [[461.11, -32.96, 182.76], [0.087605, 0.701659, 0.707062, 0.007918], [0,0,0,0], [9E9, 9E9, 9E9, 9E9, 9E9, 9E9]];
	VAR robtarget Openhole_1658 := [[460.13, -34.45, 182.78], [0.089295, 0.701446, 0.706921, 0.016229], [0,0,0,0], [9E9, 9E9, 9E9, 9E9, 9E9, 9E9]];
	VAR robtarget Openhole_1659 := [[452.05, -36.86, 181.65], [0.070349, 0.703599, 0.705208, 0.05178], [0,0,0,0], [9E9, 9E9, 9E9, 9E9, 9E9, 9E9]];
	VAR robtarget Openhole_1660 := [[451.58, -36.98, 181.57], [0.06915, 0.703717, 0.705056, 0.053818], [0,0,0,0], [9E9, 9E9, 9E9, 9E9, 9E9, 9E9]];
	VAR robtarget Openhole_1661 := [[451.1, -37.12, 181.49], [0.067993, 0.70383, 0.704895, 0.055878], [0,0,0,0], [9E9, 9E9, 9E9, 9E9, 9E9, 9E9]];
	VAR robtarget Openhole_1662 := [[450.62, -37.23, 181.4], [0.066755, 0.703949, 0.704733, 0.057889], [0,0,0,0], [9E9, 9E9, 9E9, 9E9, 9E9, 9E9]];
	VAR robtarget Openhole_1663 := [[450.15, -37.36, 181.32], [0.065576, 0.704059, 0.704562, 0.059933], [0,0,0,0], [9E9, 9E9, 9E9, 9E9, 9E9, 9E9]];
	VAR robtarget Openhole_1664 := [[449.18, -37.57, 181.15], [0.062982, 0.704296, 0.704216, 0.063874], [0,0,0,0], [9E9, 9E9, 9E9, 9E9, 9E9, 9E9]];
	VAR robtarget Openhole_1665 := [[448.69, -37.57, 181.06], [0.061339, 0.704441, 0.704061, 0.065565], [0,0,0,0], [9E9, 9E9, 9E9, 9E9, 9E9, 9E9]];
	VAR robtarget Openhole_1666 := [[448.2, -37.57, 180.98], [0.05965, 0.704586, 0.703905, 0.067211], [0,0,0,0], [9E9, 9E9, 9E9, 9E9, 9E9, 9E9]];
	VAR robtarget Openhole_1667 := [[447.24, -37.35, 180.81], [0.055674, 0.704912, 0.703658, 0.069751], [0,0,0,0], [9E9, 9E9, 9E9, 9E9, 9E9, 9E9]];
	VAR robtarget Openhole_1668 := [[446.78, -37.17, 180.73], [0.053512, 0.705079, 0.703564, 0.070694], [0,0,0,0], [9E9, 9E9, 9E9, 9E9, 9E9, 9E9]];
	VAR robtarget Openhole_1669 := [[446.31, -37, 180.66], [0.051385, 0.705237, 0.70346, 0.071722], [0,0,0,0], [9E9, 9E9, 9E9, 9E9, 9E9, 9E9]];
	VAR robtarget Openhole_1670 := [[445.84, -36.87, 180.58], [0.049313, 0.705385, 0.703343, 0.072859], [0,0,0,0], [9E9, 9E9, 9E9, 9E9, 9E9, 9E9]];
	VAR robtarget Openhole_1671 := [[443.91, -36.44, 180.27], [0.041336, 0.705898, 0.702798, 0.077938], [0,0,0,0], [9E9, 9E9, 9E9, 9E9, 9E9, 9E9]];
	VAR robtarget Openhole_1672 := [[442.94, -36.26, 180.12], [0.037412, 0.706116, 0.702501, 0.080575], [0,0,0,0], [9E9, 9E9, 9E9, 9E9, 9E9, 9E9]];
	VAR robtarget Openhole_1673 := [[441.96, -36.1, 179.97], [0.033561, 0.70631, 0.702182, 0.083311], [0,0,0,0], [9E9, 9E9, 9E9, 9E9, 9E9, 9E9]];
	VAR robtarget Openhole_1674 := [[440.98, -35.98, 179.82], [0.029793, 0.706479, 0.701839, 0.086151], [0,0,0,0], [9E9, 9E9, 9E9, 9E9, 9E9, 9E9]];
	VAR robtarget Openhole_1675 := [[440, -35.88, 179.67], [0.026128, 0.706624, 0.70147, 0.089105], [0,0,0,0], [9E9, 9E9, 9E9, 9E9, 9E9, 9E9]];
	VAR robtarget Openhole_1676 := [[439.01, -35.82, 179.51], [0.022557, 0.706747, 0.701076, 0.092156], [0,0,0,0], [9E9, 9E9, 9E9, 9E9, 9E9, 9E9]];
	VAR robtarget Openhole_1677 := [[438.02, -35.8, 179.35], [0.019086, 0.706849, 0.700655, 0.0953], [0,0,0,0], [9E9, 9E9, 9E9, 9E9, 9E9, 9E9]];
	VAR robtarget Openhole_1678 := [[437.03, -35.79, 179.2], [0.015699, 0.706932, 0.700211, 0.098512], [0,0,0,0], [9E9, 9E9, 9E9, 9E9, 9E9, 9E9]];
	VAR robtarget Openhole_1679 := [[431.62, -36.07, 178.28], [-0.001845, 0.707104, 0.69739, 0.116822], [0,0,0,0], [9E9, 9E9, 9E9, 9E9, 9E9, 9E9]];
	VAR robtarget Openhole_1680 := [[424.25, -36.48, 176.97], [-0.025379, 0.706651, 0.692911, 0.140975], [0,0,0,0], [9E9, 9E9, 9E9, 9E9, 9E9, 9E9]];
	VAR robtarget Openhole_1681 := [[421.78, -36.5, 176.55], [-0.033495, 0.706313, 0.69135, 0.148444], [0,0,0,0], [9E9, 9E9, 9E9, 9E9, 9E9, 9E9]];
	VAR robtarget Openhole_1682 := [[421.29, -36.5, 176.47], [-0.035141, 0.706233, 0.691037, 0.149895], [0,0,0,0], [9E9, 9E9, 9E9, 9E9, 9E9, 9E9]];
	VAR robtarget Openhole_1683 := [[415.86, -36.27, 175.63], [-0.053632, 0.70507, 0.687601, 0.16494], [0,0,0,0], [9E9, 9E9, 9E9, 9E9, 9E9, 9E9]];
	VAR robtarget Openhole_1684 := [[409.94, -35.68, 174.87], [-0.074298, 0.703193, 0.683915, 0.179611], [0,0,0,0], [9E9, 9E9, 9E9, 9E9, 9E9, 9E9]];
	VAR robtarget Openhole_1685 := [[403.54, -34.74, 174.26], [-0.096812, 0.700448, 0.680058, 0.193703], [0,0,0,0], [9E9, 9E9, 9E9, 9E9, 9E9, 9E9]];
	VAR robtarget Openhole_1686 := [[399.12, -33.92, 173.98], [-0.112287, 0.698134, 0.677502, 0.202463], [0,0,0,0], [9E9, 9E9, 9E9, 9E9, 9E9, 9E9]];
	VAR robtarget Openhole_1687 := [[389.32, -33.92, 172.58], [-0.139669, 0.693176, 0.670168, 0.225555], [0,0,0,0], [9E9, 9E9, 9E9, 9E9, 9E9, 9E9]];
	VAR robtarget Openhole_1688 := [[361.72, -33.92, 172.66], [-0.183051, 0.683002, 0.683002, 0.183051], [0,0,0,0], [9E9, 9E9, 9E9, 9E9, 9E9, 9E9]];
	VAR robtarget Openhole_1689 := [[362.36, -10.64, 186.11], [-0.183051, 0.683002, 0.683002, 0.183051], [0,0,0,0], [9E9, 9E9, 9E9, 9E9, 9E9, 9E9]];
	VAR robtarget Openhole_1690 := [[389.36, -10.64, 186.02], [-0.205865, 0.676476, 0.688822, 0.159765], [0,0,0,0], [9E9, 9E9, 9E9, 9E9, 9E9, 9E9]];
	VAR robtarget Openhole_1691 := [[394.36, -10.64, 185.62], [-0.193811, 0.680027, 0.691744, 0.146594], [0,0,0,0], [9E9, 9E9, 9E9, 9E9, 9E9, 9E9]];
	VAR robtarget Openhole_1692 := [[407.75, -10.06, 184.77], [-0.160415, 0.688671, 0.698996, 0.106794], [0,0,0,0], [9E9, 9E9, 9E9, 9E9, 9E9, 9E9]];
	VAR robtarget Openhole_1693 := [[423.69, -9.33, 183.58], [-0.115814, 0.697558, 0.705003, 0.054511], [0,0,0,0], [9E9, 9E9, 9E9, 9E9, 9E9, 9E9]];
	VAR robtarget Openhole_1694 := [[437.6, -8.31, 182.39], [-0.074497, 0.703172, 0.707092, 0.00463], [0,0,0,0], [9E9, 9E9, 9E9, 9E9, 9E9, 9E9]];
	VAR robtarget Openhole_1695 := [[444.02, -7.49, 181.77], [-0.055826, 0.7049, 0.706824, -0.020003], [0,0,0,0], [9E9, 9E9, 9E9, 9E9, 9E9, 9E9]];
	VAR robtarget Openhole_1696 := [[444.51, -7.43, 181.72], [-0.054357, 0.705014, 0.706768, -0.021884], [0,0,0,0], [9E9, 9E9, 9E9, 9E9, 9E9, 9E9]];
	VAR robtarget Openhole_1697 := [[445.5, -7.33, 181.61], [-0.051353, 0.70524, 0.706643, -0.025594], [0,0,0,0], [9E9, 9E9, 9E9, 9E9, 9E9, 9E9]];
	VAR robtarget Openhole_1698 := [[446.49, -7.27, 181.5], [-0.048226, 0.70546, 0.706504, -0.029201], [0,0,0,0], [9E9, 9E9, 9E9, 9E9, 9E9, 9E9]];
	VAR robtarget Openhole_1699 := [[447.49, -7.25, 181.39], [-0.044929, 0.705678, 0.706352, -0.032654], [0,0,0,0], [9E9, 9E9, 9E9, 9E9, 9E9, 9E9]];
	VAR robtarget Openhole_1700 := [[448.48, -7.26, 181.28], [-0.041525, 0.705886, 0.70619, -0.036003], [0,0,0,0], [9E9, 9E9, 9E9, 9E9, 9E9, 9E9]];
	VAR robtarget Openhole_1701 := [[452.45, -7.48, 180.84], [-0.027283, 0.70658, 0.705425, -0.048735], [0,0,0,0], [9E9, 9E9, 9E9, 9E9, 9E9, 9E9]];
	VAR robtarget Openhole_1702 := [[455.43, -7.61, 180.51], [-0.016684, 0.70691, 0.704696, -0.058344], [0,0,0,0], [9E9, 9E9, 9E9, 9E9, 9E9, 9E9]];
	VAR robtarget Openhole_1703 := [[457.42, -7.57, 180.29], [-0.010056, 0.707035, 0.704099, -0.065153], [0,0,0,0], [9E9, 9E9, 9E9, 9E9, 9E9, 9E9]];
	VAR robtarget Openhole_1704 := [[460.88, -7.27, 179.88], [0.000749, 0.707106, 0.702831, -0.077648], [0,0,0,0], [9E9, 9E9, 9E9, 9E9, 9E9, 9E9]];
	VAR robtarget Openhole_1705 := [[471.16, -5.77, 178.4], [0.03046, 0.70645, 0.697564, -0.115776], [0,0,0,0], [9E9, 9E9, 9E9, 9E9, 9E9, 9E9]];
	VAR robtarget Openhole_1706 := [[474.12, -5.49, 177.95], [0.039342, 0.706011, 0.695813, -0.125874], [0,0,0,0], [9E9, 9E9, 9E9, 9E9, 9E9, 9E9]];
	VAR robtarget Openhole_1707 := [[480.82, -3.88, 176.59], [0.056052, 0.704882, 0.69077, -0.151121], [0,0,0,0], [9E9, 9E9, 9E9, 9E9, 9E9, 9E9]];
	VAR robtarget Openhole_1708 := [[478.84, -3.85, 176.87], [0.049541, 0.705369, 0.692002, -0.145374], [0,0,0,0], [9E9, 9E9, 9E9, 9E9, 9E9, 9E9]];
	VAR robtarget Openhole_1709 := [[478.34, -3.86, 176.95], [0.047932, 0.70548, 0.69231, -0.143899], [0,0,0,0], [9E9, 9E9, 9E9, 9E9, 9E9, 9E9]];
	VAR robtarget Openhole_1710 := [[472.91, -4.06, 177.78], [0.030681, 0.706441, 0.695651, -0.126765], [0,0,0,0], [9E9, 9E9, 9E9, 9E9, 9E9, 9E9]];
	VAR robtarget Openhole_1711 := [[464.07, -4.96, 179.19], [0.003887, 0.707096, 0.700592, -0.095765], [0,0,0,0], [9E9, 9E9, 9E9, 9E9, 9E9, 9E9]];
	VAR robtarget Openhole_1712 := [[459.62, -5.2, 179.81], [-0.010432, 0.70703, 0.702526, -0.080361], [0,0,0,0], [9E9, 9E9, 9E9, 9E9, 9E9, 9E9]];
	VAR robtarget Openhole_1713 := [[459.13, -5.2, 179.88], [-0.012115, 0.707003, 0.702712, -0.078712], [0,0,0,0], [9E9, 9E9, 9E9, 9E9, 9E9, 9E9]];
	VAR robtarget Openhole_1714 := [[458.63, -5.19, 179.94], [-0.013841, 0.706971, 0.702891, -0.077102], [0,0,0,0], [9E9, 9E9, 9E9, 9E9, 9E9, 9E9]];
	VAR robtarget Openhole_1715 := [[454.68, -4.82, 180.45], [-0.028557, 0.70653, 0.7041, -0.06514], [0,0,0,0], [9E9, 9E9, 9E9, 9E9, 9E9, 9E9]];
	VAR robtarget Openhole_1716 := [[450.77, -4.2, 180.98], [-0.043982, 0.705738, 0.705042, -0.054], [0,0,0,0], [9E9, 9E9, 9E9, 9E9, 9E9, 9E9]];
	VAR robtarget Openhole_1717 := [[449.78, -4.1, 181.12], [-0.047668, 0.705498, 0.705265, -0.050997], [0,0,0,0], [9E9, 9E9, 9E9, 9E9, 9E9, 9E9]];
	VAR robtarget Openhole_1718 := [[448.79, -4.06, 181.26], [-0.051148, 0.705255, 0.705492, -0.047758], [0,0,0,0], [9E9, 9E9, 9E9, 9E9, 9E9, 9E9]];
	VAR robtarget Openhole_1719 := [[448.3, -4.06, 181.33], [-0.052824, 0.705131, 0.705604, -0.046074], [0,0,0,0], [9E9, 9E9, 9E9, 9E9, 9E9, 9E9]];
	VAR robtarget Openhole_1720 := [[447.8, -4.1, 181.4], [-0.054361, 0.705014, 0.70572, -0.044259], [0,0,0,0], [9E9, 9E9, 9E9, 9E9, 9E9, 9E9]];
	VAR robtarget Openhole_1721 := [[447.31, -4.15, 181.47], [-0.055864, 0.704897, 0.705833, -0.042416], [0,0,0,0], [9E9, 9E9, 9E9, 9E9, 9E9, 9E9]];
	VAR robtarget Openhole_1722 := [[446.82, -4.21, 181.54], [-0.057308, 0.704781, 0.705944, -0.040527], [0,0,0,0], [9E9, 9E9, 9E9, 9E9, 9E9, 9E9]];
	VAR robtarget Openhole_1723 := [[446.33, -4.29, 181.61], [-0.058708, 0.704665, 0.706052, -0.038603], [0,0,0,0], [9E9, 9E9, 9E9, 9E9, 9E9, 9E9]];
	VAR robtarget Openhole_1724 := [[445.84, -4.38, 181.68], [-0.060071, 0.704551, 0.706156, -0.036654], [0,0,0,0], [9E9, 9E9, 9E9, 9E9, 9E9, 9E9]];
	VAR robtarget Openhole_1725 := [[444.87, -4.57, 181.8], [-0.062689, 0.704322, 0.706351, -0.032678], [0,0,0,0], [9E9, 9E9, 9E9, 9E9, 9E9, 9E9]];
	VAR robtarget Openhole_1726 := [[438.56, -5.94, 182.54], [-0.079202, 0.702657, 0.707076, -0.006556], [0,0,0,0], [9E9, 9E9, 9E9, 9E9, 9E9, 9E9]];
	VAR robtarget Openhole_1727 := [[432.17, -6.93, 183.18], [-0.096813, 0.700448, 0.706867, 0.018425], [0,0,0,0], [9E9, 9E9, 9E9, 9E9, 9E9, 9E9]];
	VAR robtarget Openhole_1728 := [[431.68, -6.99, 183.23], [-0.0982, 0.700255, 0.706815, 0.020296], [0,0,0,0], [9E9, 9E9, 9E9, 9E9, 9E9, 9E9]];
	VAR robtarget Openhole_1729 := [[437.22, -4.54, 182.87], [-0.088248, 0.701578, 0.707075, -0.006666], [0,0,0,0], [9E9, 9E9, 9E9, 9E9, 9E9, 9E9]];
	VAR robtarget Openhole_1730 := [[442.5, -3.16, 182.23], [-0.075318, 0.703084, 0.706499, -0.029311], [0,0,0,0], [9E9, 9E9, 9E9, 9E9, 9E9, 9E9]];
	VAR robtarget Openhole_1731 := [[444.89, -2.47, 181.89], [-0.069605, 0.703673, 0.70599, -0.039722], [0,0,0,0], [9E9, 9E9, 9E9, 9E9, 9E9, 9E9]];
	VAR robtarget Openhole_1732 := [[445.84, -2.22, 181.75], [-0.067197, 0.703907, 0.705748, -0.043811], [0,0,0,0], [9E9, 9E9, 9E9, 9E9, 9E9, 9E9]];
	VAR robtarget Openhole_1733 := [[446.81, -2.01, 181.6], [-0.064635, 0.704147, 0.705489, -0.047802], [0,0,0,0], [9E9, 9E9, 9E9, 9E9, 9E9, 9E9]];
	VAR robtarget Openhole_1734 := [[447.3, -1.93, 181.52], [-0.063281, 0.704269, 0.705355, -0.049746], [0,0,0,0], [9E9, 9E9, 9E9, 9E9, 9E9, 9E9]];
	VAR robtarget Openhole_1735 := [[447.78, -1.85, 181.44], [-0.061883, 0.704394, 0.705217, -0.051659], [0,0,0,0], [9E9, 9E9, 9E9, 9E9, 9E9, 9E9]];
	VAR robtarget Openhole_1736 := [[448.27, -1.79, 181.36], [-0.060433, 0.70452, 0.705078, -0.05353], [0,0,0,0], [9E9, 9E9, 9E9, 9E9, 9E9, 9E9]];
	VAR robtarget Openhole_1737 := [[448.77, -1.75, 181.28], [-0.058886, 0.704651, 0.704939, -0.055324], [0,0,0,0], [9E9, 9E9, 9E9, 9E9, 9E9, 9E9]];
	VAR robtarget Openhole_1738 := [[449.26, -1.74, 181.2], [-0.057252, 0.704785, 0.704803, -0.057039], [0,0,0,0], [9E9, 9E9, 9E9, 9E9, 9E9, 9E9]];
	VAR robtarget Openhole_1739 := [[449.75, -1.74, 181.11], [-0.055569, 0.70492, 0.704666, -0.058702], [0,0,0,0], [9E9, 9E9, 9E9, 9E9, 9E9, 9E9]];
	VAR robtarget Openhole_1740 := [[450.24, -1.78, 181.03], [-0.053771, 0.705059, 0.704536, -0.060243], [0,0,0,0], [9E9, 9E9, 9E9, 9E9, 9E9, 9E9]];
	VAR robtarget Openhole_1741 := [[450.73, -1.83, 180.95], [-0.051934, 0.705197, 0.704407, -0.061735], [0,0,0,0], [9E9, 9E9, 9E9, 9E9, 9E9, 9E9]];
	VAR robtarget Openhole_1742 := [[451.22, -1.9, 180.87], [-0.050044, 0.705334, 0.70428, -0.063163], [0,0,0,0], [9E9, 9E9, 9E9, 9E9, 9E9, 9E9]];
	VAR robtarget Openhole_1743 := [[456.58, -2.86, 180.06], [-0.028614, 0.706528, 0.702792, -0.077993], [0,0,0,0], [9E9, 9E9, 9E9, 9E9, 9E9, 9E9]];
	VAR robtarget Openhole_1744 := [[458.54, -3.07, 179.77], [-0.02118, 0.706789, 0.702121, -0.083825], [0,0,0,0], [9E9, 9E9, 9E9, 9E9, 9E9, 9E9]];
	VAR robtarget Openhole_1745 := [[459.53, -3.13, 179.62], [-0.01762, 0.706887, 0.701746, -0.086906], [0,0,0,0], [9E9, 9E9, 9E9, 9E9, 9E9, 9E9]];
	VAR robtarget Openhole_1746 := [[460.52, -3.16, 179.47], [-0.014158, 0.706965, 0.701346, -0.090078], [0,0,0,0], [9E9, 9E9, 9E9, 9E9, 9E9, 9E9]];
	VAR robtarget Openhole_1747 := [[461.01, -3.16, 179.4], [-0.012469, 0.706997, 0.701135, -0.091701], [0,0,0,0], [9E9, 9E9, 9E9, 9E9, 9E9, 9E9]];
	VAR robtarget Openhole_1748 := [[461.51, -3.15, 179.32], [-0.010789, 0.707024, 0.700921, -0.093327], [0,0,0,0], [9E9, 9E9, 9E9, 9E9, 9E9, 9E9]];
	VAR robtarget Openhole_1749 := [[466.44, -2.87, 178.52], [0.005021, 0.707089, 0.698464, -0.110219], [0,0,0,0], [9E9, 9E9, 9E9, 9E9, 9E9, 9E9]];
	VAR robtarget Openhole_1750 := [[473.81, -2.37, 177.26], [0.0282, 0.706544, 0.694118, -0.134911], [0,0,0,0], [9E9, 9E9, 9E9, 9E9, 9E9, 9E9]];
	VAR robtarget Openhole_1751 := [[476.77, -2.31, 176.77], [0.037825, 0.706094, 0.692279, -0.14405], [0,0,0,0], [9E9, 9E9, 9E9, 9E9, 9E9, 9E9]];
	VAR robtarget Openhole_1752 := [[477.26, -2.32, 176.69], [0.039458, 0.706005, 0.691971, -0.145521], [0,0,0,0], [9E9, 9E9, 9E9, 9E9, 9E9, 9E9]];
	VAR robtarget Openhole_1753 := [[482.7, -2.51, 175.88], [0.057758, 0.704744, 0.688574, -0.16083], [0,0,0,0], [9E9, 9E9, 9E9, 9E9, 9E9, 9E9]];
	VAR robtarget Openhole_1754 := [[489.12, -3.09, 175.08], [0.079837, 0.702585, 0.684584, -0.177046], [0,0,0,0], [9E9, 9E9, 9E9, 9E9, 9E9, 9E9]];
	VAR robtarget Openhole_1755 := [[495.54, -3.95, 174.47], [0.101905, 0.699725, 0.680674, -0.191527], [0,0,0,0], [9E9, 9E9, 9E9, 9E9, 9E9, 9E9]];
	VAR robtarget Openhole_1756 := [[495.59, -2.66, 173.89], [0.098193, 0.700256, 0.679563, -0.195434], [0,0,0,0], [9E9, 9E9, 9E9, 9E9, 9E9, 9E9]];
	VAR robtarget Openhole_1757 := [[489.19, -1.71, 174.53], [0.075787, 0.703034, 0.683441, -0.181407], [0,0,0,0], [9E9, 9E9, 9E9, 9E9, 9E9, 9E9]];
	VAR robtarget Openhole_1758 := [[483.28, -1.11, 175.33], [0.055214, 0.704948, 0.687155, -0.166787], [0,0,0,0], [9E9, 9E9, 9E9, 9E9, 9E9, 9E9]];
	VAR robtarget Openhole_1759 := [[477.85, -0.87, 176.2], [0.036772, 0.70615, 0.690618, -0.15181], [0,0,0,0], [9E9, 9E9, 9E9, 9E9, 9E9, 9E9]];
	VAR robtarget Openhole_1760 := [[476.87, -0.86, 176.37], [0.033499, 0.706313, 0.691251, -0.148903], [0,0,0,0], [9E9, 9E9, 9E9, 9E9, 9E9, 9E9]];
	VAR robtarget Openhole_1761 := [[476.37, -0.86, 176.45], [0.031874, 0.706388, 0.691567, -0.147428], [0,0,0,0], [9E9, 9E9, 9E9, 9E9, 9E9, 9E9]];
	VAR robtarget Openhole_1762 := [[470.48, -1.08, 177.53], [0.01284, 0.70699, 0.695288, -0.128744], [0,0,0,0], [9E9, 9E9, 9E9, 9E9, 9E9, 9E9]];
	VAR robtarget Openhole_1763 := [[462.62, -1.59, 178.95], [-0.012155, 0.707002, 0.6997, -0.102076], [0,0,0,0], [9E9, 9E9, 9E9, 9E9, 9E9, 9E9]];
	VAR robtarget Openhole_1764 := [[461.64, -1.61, 179.12], [-0.015439, 0.706938, 0.700172, -0.098785], [0,0,0,0], [9E9, 9E9, 9E9, 9E9, 9E9, 9E9]];
	VAR robtarget Openhole_1765 := [[461.14, -1.61, 179.2], [-0.017116, 0.7069, 0.700399, -0.097167], [0,0,0,0], [9E9, 9E9, 9E9, 9E9, 9E9, 9E9]];
	VAR robtarget Openhole_1766 := [[460.65, -1.61, 179.29], [-0.018811, 0.706857, 0.70062, -0.095561], [0,0,0,0], [9E9, 9E9, 9E9, 9E9, 9E9, 9E9]];
	VAR robtarget Openhole_1767 := [[460.16, -1.6, 179.37], [-0.020529, 0.706809, 0.700834, -0.093974], [0,0,0,0], [9E9, 9E9, 9E9, 9E9, 9E9, 9E9]];
	VAR robtarget Openhole_1768 := [[459.17, -1.56, 179.53], [-0.024048, 0.706698, 0.701243, -0.090875], [0,0,0,0], [9E9, 9E9, 9E9, 9E9, 9E9, 9E9]];
	VAR robtarget Openhole_1769 := [[457.2, -1.38, 179.85], [-0.031369, 0.706411, 0.701984, -0.084958], [0,0,0,0], [9E9, 9E9, 9E9, 9E9, 9E9, 9E9]];
	VAR robtarget Openhole_1770 := [[454.77, -0.99, 180.24], [-0.040968, 0.705919, 0.702783, -0.078081], [0,0,0,0], [9E9, 9E9, 9E9, 9E9, 9E9, 9E9]];
	VAR robtarget Openhole_1771 := [[453.8, -0.8, 180.4], [-0.044907, 0.705679, 0.703068, -0.075466], [0,0,0,0], [9E9, 9E9, 9E9, 9E9, 9E9, 9E9]];
	VAR robtarget Openhole_1772 := [[452.84, -0.58, 180.56], [-0.048916, 0.705413, 0.703333, -0.07296], [0,0,0,0], [9E9, 9E9, 9E9, 9E9, 9E9, 9E9]];
	VAR robtarget Openhole_1773 := [[451.9, -0.27, 180.72], [-0.053123, 0.705108, 0.703553, -0.070807], [0,0,0,0], [9E9, 9E9, 9E9, 9E9, 9E9, 9E9]];
	VAR robtarget Openhole_1774 := [[451.43, -0.1, 180.8], [-0.055254, 0.704945, 0.703654, -0.069793], [0,0,0,0], [9E9, 9E9, 9E9, 9E9, 9E9, 9E9]];
	VAR robtarget Openhole_1775 := [[450.48, 0.12, 180.97], [-0.059263, 0.704619, 0.703896, -0.067304], [0,0,0,0], [9E9, 9E9, 9E9, 9E9, 9E9, 9E9]];
	VAR robtarget Openhole_1776 := [[449.49, 0.16, 181.15], [-0.062713, 0.70432, 0.704197, -0.064088], [0,0,0,0], [9E9, 9E9, 9E9, 9E9, 9E9, 9E9]];
	VAR robtarget Openhole_1777 := [[448.52, 0, 181.33], [-0.065478, 0.704069, 0.704534, -0.060265], [0,0,0,0], [9E9, 9E9, 9E9, 9E9, 9E9, 9E9]];
	VAR robtarget Openhole_1778 := [[448.04, -0.13, 181.42], [-0.066675, 0.703956, 0.704705, -0.058232], [0,0,0,0], [9E9, 9E9, 9E9, 9E9, 9E9, 9E9]];
	VAR robtarget Openhole_1779 := [[447.57, -0.24, 181.5], [-0.067906, 0.703839, 0.704868, -0.056217], [0,0,0,0], [9E9, 9E9, 9E9, 9E9, 9E9, 9E9]];
	VAR robtarget Openhole_1780 := [[447.09, -0.38, 181.59], [-0.069056, 0.703727, 0.70503, -0.054154], [0,0,0,0], [9E9, 9E9, 9E9, 9E9, 9E9, 9E9]];
	VAR robtarget Openhole_1781 := [[446.14, -0.63, 181.75], [-0.071439, 0.703489, 0.705332, -0.05007], [0,0,0,0], [9E9, 9E9, 9E9, 9E9, 9E9, 9E9]];
	VAR robtarget Openhole_1782 := [[445.19, -0.91, 181.91], [-0.073741, 0.703251, 0.705613, -0.045935], [0,0,0,0], [9E9, 9E9, 9E9, 9E9, 9E9, 9E9]];
	VAR robtarget Openhole_1783 := [[439.03, -2.77, 182.8], [-0.08811, 0.701596, 0.70686, -0.018684], [0,0,0,0], [9E9, 9E9, 9E9, 9E9, 9E9, 9E9]];
	VAR robtarget Openhole_1784 := [[441.88, -4.7, 182.21], [-0.072287, 0.703402, 0.706764, -0.022025], [0,0,0,0], [9E9, 9E9, 9E9, 9E9, 9E9, 9E9]];
	VAR robtarget Openhole_1785 := [[444.74, -6.64, 181.73], [-0.056229, 0.704868, 0.706653, -0.02533], [0,0,0,0], [9E9, 9E9, 9E9, 9E9, 9E9, 9E9]];
	VAR robtarget Openhole_1786 := [[445.23, -6.56, 181.67], [-0.054825, 0.704978, 0.706581, -0.02726], [0,0,0,0], [9E9, 9E9, 9E9, 9E9, 9E9, 9E9]];
	VAR robtarget Openhole_1787 := [[446.22, -6.44, 181.56], [-0.051917, 0.705198, 0.706425, -0.031042], [0,0,0,0], [9E9, 9E9, 9E9, 9E9, 9E9, 9E9]];
	VAR robtarget Openhole_1788 := [[447.21, -6.37, 181.44], [-0.048803, 0.705421, 0.706257, -0.034655], [0,0,0,0], [9E9, 9E9, 9E9, 9E9, 9E9, 9E9]];
	VAR robtarget Openhole_1789 := [[447.71, -6.35, 181.38], [-0.047174, 0.705531, 0.706169, -0.036397], [0,0,0,0], [9E9, 9E9, 9E9, 9E9, 9E9, 9E9]];
	VAR robtarget Openhole_1790 := [[448.2, -6.35, 181.32], [-0.045514, 0.70564, 0.706079, -0.038109], [0,0,0,0], [9E9, 9E9, 9E9, 9E9, 9E9, 9E9]];
	VAR robtarget Openhole_1791 := [[449.69, -6.4, 181.14], [-0.040277, 0.705959, 0.705799, -0.042986], [0,0,0,0], [9E9, 9E9, 9E9, 9E9, 9E9, 9E9]];
	VAR robtarget Openhole_1792 := [[452.66, -6.67, 180.79], [-0.029284, 0.7065, 0.705181, -0.05215], [0,0,0,0], [9E9, 9E9, 9E9, 9E9, 9E9, 9E9]];
	VAR robtarget Openhole_1793 := [[453.65, -6.78, 180.67], [-0.025533, 0.706646, 0.704957, -0.055097], [0,0,0,0], [9E9, 9E9, 9E9, 9E9, 9E9, 9E9]];
	VAR robtarget Openhole_1794 := [[454.64, -6.86, 180.56], [-0.021894, 0.706768, 0.70471, -0.058175], [0,0,0,0], [9E9, 9E9, 9E9, 9E9, 9E9, 9E9]];
	VAR robtarget Openhole_1795 := [[457.01, -8.37, 180.4], [-0.008773, 0.707052, 0.704462, -0.061101], [0,0,0,0], [9E9, 9E9, 9E9, 9E9, 9E9, 9E9]];
	VAR robtarget Openhole_1796 := [[455.02, -8.48, 180.61], [-0.015165, 0.706944, 0.705038, -0.054055], [0,0,0,0], [9E9, 9E9, 9E9, 9E9, 9E9, 9E9]];
	VAR robtarget Openhole_1797 := [[454.03, -8.5, 180.71], [-0.018491, 0.706865, 0.705291, -0.050637], [0,0,0,0], [9E9, 9E9, 9E9, 9E9, 9E9, 9E9]];
	VAR robtarget Openhole_1798 := [[453.53, -8.5, 180.76], [-0.020191, 0.706818, 0.70541, -0.048961], [0,0,0,0], [9E9, 9E9, 9E9, 9E9, 9E9, 9E9]];
	VAR robtarget Openhole_1799 := [[453.03, -8.5, 180.81], [-0.02187, 0.706768, 0.705525, -0.047265], [0,0,0,0], [9E9, 9E9, 9E9, 9E9, 9E9, 9E9]];
	VAR robtarget Openhole_1800 := [[452.53, -8.5, 180.86], [-0.023559, 0.706714, 0.705637, -0.045574], [0,0,0,0], [9E9, 9E9, 9E9, 9E9, 9E9, 9E9]];
	VAR robtarget Openhole_1801 := [[452.04, -8.5, 180.91], [-0.02526, 0.706655, 0.705743, -0.043896], [0,0,0,0], [9E9, 9E9, 9E9, 9E9, 9E9, 9E9]];
	VAR robtarget Openhole_1802 := [[447.06, -8.37, 181.42], [-0.042597, 0.705823, 0.706575, -0.02743], [0,0,0,0], [9E9, 9E9, 9E9, 9E9, 9E9, 9E9]];
	VAR robtarget Openhole_1803 := [[446.57, -8.37, 181.47], [-0.044292, 0.705718, 0.706638, -0.025744], [0,0,0,0], [9E9, 9E9, 9E9, 9E9, 9E9, 9E9]];
	VAR robtarget Openhole_1804 := [[446.07, -8.37, 181.52], [-0.04596, 0.705612, 0.706698, -0.024034], [0,0,0,0], [9E9, 9E9, 9E9, 9E9, 9E9, 9E9]];
	VAR robtarget Openhole_1805 := [[445.07, -8.4, 181.62], [-0.04923, 0.705391, 0.706808, -0.020551], [0,0,0,0], [9E9, 9E9, 9E9, 9E9, 9E9, 9E9]];
	VAR robtarget Openhole_1806 := [[444.58, -8.42, 181.67], [-0.050818, 0.705278, 0.706858, -0.018767], [0,0,0,0], [9E9, 9E9, 9E9, 9E9, 9E9, 9E9]];
	VAR robtarget Openhole_1807 := [[438.63, -8.96, 182.22], [-0.068955, 0.703737, 0.707099, 0.003308], [0,0,0,0], [9E9, 9E9, 9E9, 9E9, 9E9, 9E9]];
	VAR robtarget Openhole_1808 := [[437.22, -10.53, 182.17], [-0.068387, 0.703792, 0.706981, 0.013363], [0,0,0,0], [9E9, 9E9, 9E9, 9E9, 9E9, 9E9]];
	VAR robtarget Openhole_1809 := [[437.71, -10.53, 182.13], [-0.066719, 0.703952, 0.70701, 0.011691], [0,0,0,0], [9E9, 9E9, 9E9, 9E9, 9E9, 9E9]];
	VAR robtarget Openhole_1810 := [[438.21, -10.53, 182.09], [-0.065064, 0.704107, 0.707036, 0.01], [0,0,0,0], [9E9, 9E9, 9E9, 9E9, 9E9, 9E9]];
	VAR robtarget Openhole_1811 := [[438.71, -10.53, 182.05], [-0.063401, 0.704259, 0.707058, 0.008315], [0,0,0,0], [9E9, 9E9, 9E9, 9E9, 9E9, 9E9]];
	VAR robtarget Openhole_1812 := [[439.21, -10.53, 182.01], [-0.061739, 0.704406, 0.707076, 0.006623], [0,0,0,0], [9E9, 9E9, 9E9, 9E9, 9E9, 9E9]];
	VAR robtarget Openhole_1813 := [[439.71, -10.53, 181.97], [-0.060087, 0.704549, 0.70709, 0.00492], [0,0,0,0], [9E9, 9E9, 9E9, 9E9, 9E9, 9E9]];
	VAR robtarget Openhole_1814 := [[442.7, -10.49, 181.73], [-0.050196, 0.705323, 0.707086, -0.005389], [0,0,0,0], [9E9, 9E9, 9E9, 9E9, 9E9, 9E9]];
	VAR robtarget Openhole_1815 := [[443.69, -10.51, 181.64], [-0.046774, 0.705558, 0.707053, -0.008718], [0,0,0,0], [9E9, 9E9, 9E9, 9E9, 9E9, 9E9]];
	VAR robtarget Openhole_1816 := [[444.19, -10.54, 181.6], [-0.044998, 0.705674, 0.707032, -0.010315], [0,0,0,0], [9E9, 9E9, 9E9, 9E9, 9E9, 9E9]];
	VAR robtarget Openhole_1817 := [[444.69, -10.59, 181.56], [-0.043151, 0.705789, 0.707008, -0.01183], [0,0,0,0], [9E9, 9E9, 9E9, 9E9, 9E9, 9E9]];
	VAR robtarget Openhole_1818 := [[445.18, -10.67, 181.52], [-0.041216, 0.705905, 0.706983, -0.013231], [0,0,0,0], [9E9, 9E9, 9E9, 9E9, 9E9, 9E9]];
	VAR robtarget Openhole_1819 := [[446.16, -10.86, 181.43], [-0.037284, 0.706123, 0.706927, -0.015951], [0,0,0,0], [9E9, 9E9, 9E9, 9E9, 9E9, 9E9]];
	VAR robtarget Openhole_1820 := [[446.72, -11.14, 181.38], [-0.034413, 0.706269, 0.706905, -0.01688], [0,0,0,0], [9E9, 9E9, 9E9, 9E9, 9E9, 9E9]];
	VAR robtarget Openhole_1821 := [[453.3, -11.75, 180.9], [-0.009977, 0.707036, 0.706126, -0.037234], [0,0,0,0], [9E9, 9E9, 9E9, 9E9, 9E9, 9E9]];
	VAR robtarget Openhole_1822 := [[453.93, -11.26, 180.84], [-0.009479, 0.707043, 0.705918, -0.040991], [0,0,0,0], [9E9, 9E9, 9E9, 9E9, 9E9, 9E9]];
	VAR robtarget Openhole_1823 := [[454.39, -11.08, 180.8], [-0.008542, 0.707055, 0.705787, -0.043185], [0,0,0,0], [9E9, 9E9, 9E9, 9E9, 9E9, 9E9]];
	VAR robtarget Openhole_1824 := [[454.86, -10.92, 180.75], [-0.007478, 0.707067, 0.705653, -0.045319], [0,0,0,0], [9E9, 9E9, 9E9, 9E9, 9E9, 9E9]];
	VAR robtarget Openhole_1825 := [[455.82, -10.65, 180.66], [-0.005129, 0.707088, 0.705375, -0.049463], [0,0,0,0], [9E9, 9E9, 9E9, 9E9, 9E9, 9E9]];
	VAR robtarget Openhole_1826 := [[456.31, -10.53, 180.61], [-0.003886, 0.707096, 0.705229, -0.051493], [0,0,0,0], [9E9, 9E9, 9E9, 9E9, 9E9, 9E9]];
	VAR robtarget Openhole_1827 := [[456.79, -10.4, 180.56], [-0.002682, 0.707102, 0.705077, -0.053541], [0,0,0,0], [9E9, 9E9, 9E9, 9E9, 9E9, 9E9]];
	VAR robtarget Openhole_1828 := [[457.75, -10.16, 180.46], [-0.000183, 0.707107, 0.704759, -0.057575], [0,0,0,0], [9E9, 9E9, 9E9, 9E9, 9E9, 9E9]];
	VAR robtarget Openhole_1829 := [[466.46, -8.15, 179.39], [0.022544, 0.706747, 0.700965, -0.092993], [0,0,0,0], [9E9, 9E9, 9E9, 9E9, 9E9, 9E9]];
	VAR robtarget Openhole_1830 := [[468.4, -7.76, 179.11], [0.027768, 0.706561, 0.699924, -0.100529], [0,0,0,0], [9E9, 9E9, 9E9, 9E9, 9E9, 9E9]];
	VAR robtarget Openhole_1831 := [[465.51, -9.96, 179.77], [0.025361, 0.706652, 0.70211, -0.083911], [0,0,0,0], [9E9, 9E9, 9E9, 9E9, 9E9, 9E9]];
	VAR robtarget Openhole_1832 := [[464.08, -10.39, 179.96], [0.022001, 0.706764, 0.702812, -0.07782], [0,0,0,0], [9E9, 9E9, 9E9, 9E9, 9E9, 9E9]];
	VAR robtarget Openhole_1833 := [[461.73, -11.18, 180.25], [0.016687, 0.70691, 0.703885, -0.067422], [0,0,0,0], [9E9, 9E9, 9E9, 9E9, 9E9, 9E9]];
	VAR robtarget Openhole_1834 := [[459.4, -12.06, 180.51], [0.011809, 0.707008, 0.704829, -0.056709], [0,0,0,0], [9E9, 9E9, 9E9, 9E9, 9E9, 9E9]];
	VAR robtarget Openhole_1835 := [[458.49, -12.46, 180.6], [0.01006, 0.707035, 0.705169, -0.052313], [0,0,0,0], [9E9, 9E9, 9E9, 9E9, 9E9, 9E9]];
	VAR robtarget Openhole_1836 := [[457.59, -12.89, 180.69], [0.008472, 0.707056, 0.705486, -0.047843], [0,0,0,0], [9E9, 9E9, 9E9, 9E9, 9E9, 9E9]];
	VAR robtarget Openhole_1837 := [[457.15, -13.13, 180.74], [0.007784, 0.707064, 0.705637, -0.04557], [0,0,0,0], [9E9, 9E9, 9E9, 9E9, 9E9, 9E9]];
	VAR robtarget Openhole_1838 := [[456.73, -13.4, 180.78], [0.00727, 0.707069, 0.705783, -0.043247], [0,0,0,0], [9E9, 9E9, 9E9, 9E9, 9E9, 9E9]];
	VAR robtarget Openhole_1839 := [[456.33, -13.69, 180.82], [0.006888, 0.707073, 0.705923, -0.040897], [0,0,0,0], [9E9, 9E9, 9E9, 9E9, 9E9, 9E9]];
	VAR robtarget Openhole_1840 := [[455.86, -14.06, 180.87], [0.006555, 0.707076, 0.706082, -0.03806], [0,0,0,0], [9E9, 9E9, 9E9, 9E9, 9E9, 9E9]];
	VAR robtarget Openhole_1841 := [[443.92, -12.82, 181.51], [-0.038211, 0.706074, 0.707105, -0.001666], [0,0,0,0], [9E9, 9E9, 9E9, 9E9, 9E9, 9E9]];
	VAR robtarget Openhole_1842 := [[443.19, -12.46, 181.57], [-0.041903, 0.705864, 0.707107, -0.000402], [0,0,0,0], [9E9, 9E9, 9E9, 9E9, 9E9, 9E9]];
	VAR robtarget Openhole_1843 := [[442.2, -12.35, 181.64], [-0.045615, 0.705634, 0.707102, 0.0026], [0,0,0,0], [9E9, 9E9, 9E9, 9E9, 9E9, 9E9]];
	VAR robtarget Openhole_1844 := [[441.7, -12.31, 181.68], [-0.047419, 0.705515, 0.707095, 0.004161], [0,0,0,0], [9E9, 9E9, 9E9, 9E9, 9E9, 9E9]];
	VAR robtarget Openhole_1845 := [[440.21, -12.22, 181.78], [-0.052722, 0.705139, 0.70705, 0.008948], [0,0,0,0], [9E9, 9E9, 9E9, 9E9, 9E9, 9E9]];
	VAR robtarget Openhole_1846 := [[439.21, -12.15, 181.85], [-0.056296, 0.704862, 0.707004, 0.012076], [0,0,0,0], [9E9, 9E9, 9E9, 9E9, 9E9, 9E9]];
	VAR robtarget Openhole_1847 := [[438.22, -12.1, 181.92], [-0.059804, 0.704573, 0.706942, 0.015265], [0,0,0,0], [9E9, 9E9, 9E9, 9E9, 9E9, 9E9]];
	VAR robtarget Openhole_1848 := [[435.3, -16.15, 181.57], [-0.055872, 0.704896, 0.706044, 0.038756], [0,0,0,0], [9E9, 9E9, 9E9, 9E9, 9E9, 9E9]];
	VAR robtarget Openhole_1849 := [[434.8, -16.09, 181.59], [-0.057716, 0.704747, 0.705962, 0.040217], [0,0,0,0], [9E9, 9E9, 9E9, 9E9, 9E9, 9E9]];
	VAR robtarget Openhole_1850 := [[433.81, -16, 181.63], [-0.061326, 0.704442, 0.705785, 0.04322], [0,0,0,0], [9E9, 9E9, 9E9, 9E9, 9E9, 9E9]];
	VAR robtarget Openhole_1851 := [[425.83, -15.62, 181.95], [-0.088551, 0.70154, 0.703807, 0.068235], [0,0,0,0], [9E9, 9E9, 9E9, 9E9, 9E9, 9E9]];
	VAR robtarget Openhole_1852 := [[411.84, -15.42, 182.48], [-0.132116, 0.694655, 0.698285, 0.11135], [0,0,0,0], [9E9, 9E9, 9E9, 9E9, 9E9, 9E9]];
	VAR robtarget Openhole_1853 := [[411.34, -15.42, 182.5], [-0.133579, 0.694375, 0.698044, 0.112846], [0,0,0,0], [9E9, 9E9, 9E9, 9E9, 9E9, 9E9]];
	VAR robtarget Openhole_1854 := [[410.84, -15.42, 182.52], [-0.135034, 0.694094, 0.697801, 0.114341], [0,0,0,0], [9E9, 9E9, 9E9, 9E9, 9E9, 9E9]];
	VAR robtarget Openhole_1855 := [[399.84, -15.62, 182.8], [-0.165109, 0.68756, 0.691776, 0.146444], [0,0,0,0], [9E9, 9E9, 9E9, 9E9, 9E9, 9E9]];
	VAR robtarget Openhole_1856 := [[394.35, -15.88, 182.85], [-0.178674, 0.684161, 0.688316, 0.16193], [0,0,0,0], [9E9, 9E9, 9E9, 9E9, 9E9, 9E9]];
	VAR robtarget Openhole_1857 := [[389.35, -15.88, 183], [-0.191107, 0.680792, 0.685179, 0.174728], [0,0,0,0], [9E9, 9E9, 9E9, 9E9, 9E9, 9E9]];
	VAR robtarget Openhole_1858 := [[362.35, -15.88, 183.09], [-0.183051, 0.683002, 0.683002, 0.183051], [0,0,0,0], [9E9, 9E9, 9E9, 9E9, 9E9, 9E9]];
	VAR robtarget Openhole_1859 := [[362.34, -21.09, 180.07], [-0.183051, 0.683002, 0.683002, 0.183051], [0,0,0,0], [9E9, 9E9, 9E9, 9E9, 9E9, 9E9]];
	VAR robtarget Openhole_1860 := [[389.34, -21.09, 179.99], [-0.176277, 0.684782, 0.681216, 0.189592], [0,0,0,0], [9E9, 9E9, 9E9, 9E9, 9E9, 9E9]];
	VAR robtarget Openhole_1861 := [[394.34, -21.09, 180.09], [-0.163466, 0.687953, 0.684552, 0.17717], [0,0,0,0], [9E9, 9E9, 9E9, 9E9, 9E9, 9E9]];
	VAR robtarget Openhole_1862 := [[395.21, -21.06, 180.12], [-0.161268, 0.688471, 0.685147, 0.174852], [0,0,0,0], [9E9, 9E9, 9E9, 9E9, 9E9, 9E9]];
	VAR robtarget Openhole_1863 := [[401.7, -20.78, 180.38], [-0.144509, 0.692183, 0.689478, 0.15691], [0,0,0,0], [9E9, 9E9, 9E9, 9E9, 9E9, 9E9]];
	VAR robtarget Openhole_1864 := [[406.7, -20.73, 180.48], [-0.130508, 0.694959, 0.69252, 0.142887], [0,0,0,0], [9E9, 9E9, 9E9, 9E9, 9E9, 9E9]];
	VAR robtarget Openhole_1865 := [[407.2, -20.73, 180.49], [-0.129061, 0.695229, 0.69281, 0.141471], [0,0,0,0], [9E9, 9E9, 9E9, 9E9, 9E9, 9E9]];
	VAR robtarget Openhole_1866 := [[421.2, -20.9, 180.67], [-0.085981, 0.70186, 0.699964, 0.100253], [0,0,0,0], [9E9, 9E9, 9E9, 9E9, 9E9, 9E9]];
	VAR robtarget Openhole_1867 := [[421.7, -20.9, 180.68], [-0.084396, 0.702052, 0.700186, 0.098691], [0,0,0,0], [9E9, 9E9, 9E9, 9E9, 9E9, 9E9]];
	VAR robtarget Openhole_1868 := [[425.2, -20.8, 180.77], [-0.073501, 0.703276, 0.701692, 0.087343], [0,0,0,0], [9E9, 9E9, 9E9, 9E9, 9E9, 9E9]];
	VAR robtarget Openhole_1869 := [[426.19, -20.74, 180.8], [-0.070488, 0.703585, 0.702107, 0.083942], [0,0,0,0], [9E9, 9E9, 9E9, 9E9, 9E9, 9E9]];
	VAR robtarget Openhole_1870 := [[428.18, -20.56, 180.87], [-0.064607, 0.704149, 0.702909, 0.076937], [0,0,0,0], [9E9, 9E9, 9E9, 9E9, 9E9, 9E9]];
	VAR robtarget Openhole_1871 := [[429.17, -20.43, 180.91], [-0.061789, 0.704402, 0.703297, 0.073298], [0,0,0,0], [9E9, 9E9, 9E9, 9E9, 9E9, 9E9]];
	VAR robtarget Openhole_1872 := [[429.67, -20.35, 180.93], [-0.060425, 0.70452, 0.703489, 0.071436], [0,0,0,0], [9E9, 9E9, 9E9, 9E9, 9E9, 9E9]];
	VAR robtarget Openhole_1873 := [[431.14, -20.07, 181], [-0.056514, 0.704845, 0.704049, 0.065691], [0,0,0,0], [9E9, 9E9, 9E9, 9E9, 9E9, 9E9]];
	VAR robtarget Openhole_1874 := [[433.09, -19.64, 181.09], [-0.051504, 0.705229, 0.704739, 0.057824], [0,0,0,0], [9E9, 9E9, 9E9, 9E9, 9E9, 9E9]];
	VAR robtarget Openhole_1875 := [[431.92, -18.36, 181.29], [-0.059665, 0.704585, 0.704775, 0.057375], [0,0,0,0], [9E9, 9E9, 9E9, 9E9, 9E9, 9E9]];
	VAR robtarget Openhole_1876 := [[431.42, -18.38, 181.29], [-0.061212, 0.704452, 0.704631, 0.059119], [0,0,0,0], [9E9, 9E9, 9E9, 9E9, 9E9, 9E9]];
	VAR robtarget Openhole_1877 := [[430.42, -18.38, 181.3], [-0.064502, 0.704159, 0.704348, 0.062403], [0,0,0,0], [9E9, 9E9, 9E9, 9E9, 9E9, 9E9]];
	VAR robtarget Openhole_1878 := [[426.43, -18.45, 181.31], [-0.07731, 0.702868, 0.703051, 0.075626], [0,0,0,0], [9E9, 9E9, 9E9, 9E9, 9E9, 9E9]];
	VAR robtarget Openhole_1879 := [[425.93, -18.44, 181.31], [-0.078931, 0.702688, 0.702877, 0.077228], [0,0,0,0], [9E9, 9E9, 9E9, 9E9, 9E9, 9E9]];
	VAR robtarget Openhole_1880 := [[408.43, -18.16, 181.52], [-0.133483, 0.694393, 0.695057, 0.129981], [0,0,0,0], [9E9, 9E9, 9E9, 9E9, 9E9, 9E9]];
	VAR robtarget Openhole_1881 := [[407.93, -18.16, 181.53], [-0.134925, 0.694115, 0.694785, 0.131429], [0,0,0,0], [9E9, 9E9, 9E9, 9E9, 9E9, 9E9]];
	VAR robtarget Openhole_1882 := [[398.93, -18.33, 181.52], [-0.159456, 0.688893, 0.689449, 0.157035], [0,0,0,0], [9E9, 9E9, 9E9, 9E9, 9E9, 9E9]];
	VAR robtarget Openhole_1883 := [[394.35, -18.56, 181.43], [-0.170861, 0.686153, 0.686422, 0.16978], [0,0,0,0], [9E9, 9E9, 9E9, 9E9, 9E9, 9E9]];
	VAR robtarget Openhole_1884 := [[362.35, -18.56, 181.54], [-0.183051, 0.683002, 0.683002, 0.183051], [0,0,0,0], [9E9, 9E9, 9E9, 9E9, 9E9, 9E9]];
	VAR robtarget Openhole_1885 := [[362.35, -17.6, 182.09], [-0.183051, 0.683002, 0.683002, 0.183051], [0,0,0,0], [9E9, 9E9, 9E9, 9E9, 9E9, 9E9]];
	VAR robtarget Openhole_1886 := [[389.35, -17.6, 182.01], [-0.186222, 0.682145, 0.683906, 0.179644], [0,0,0,0], [9E9, 9E9, 9E9, 9E9, 9E9, 9E9]];
	VAR robtarget Openhole_1887 := [[394.35, -17.6, 181.94], [-0.173663, 0.68545, 0.687111, 0.16697], [0,0,0,0], [9E9, 9E9, 9E9, 9E9, 9E9, 9E9]];
	VAR robtarget Openhole_1888 := [[403.05, -17.26, 181.97], [-0.151463, 0.690695, 0.692589, 0.14255], [0,0,0,0], [9E9, 9E9, 9E9, 9E9, 9E9, 9E9]];
	VAR robtarget Openhole_1889 := [[408.54, -17.2, 181.9], [-0.136132, 0.693879, 0.69567, 0.126663], [0,0,0,0], [9E9, 9E9, 9E9, 9E9, 9E9, 9E9]];
	VAR robtarget Openhole_1890 := [[409.04, -17.2, 181.89], [-0.134687, 0.694161, 0.695934, 0.125205], [0,0,0,0], [9E9, 9E9, 9E9, 9E9, 9E9, 9E9]];
	VAR robtarget Openhole_1891 := [[423.54, -17.43, 181.58], [-0.089877, 0.701372, 0.702387, 0.081559], [0,0,0,0], [9E9, 9E9, 9E9, 9E9, 9E9, 9E9]];
	VAR robtarget Openhole_1892 := [[433.04, -17.58, 181.41], [-0.058575, 0.704676, 0.705257, 0.051112], [0,0,0,0], [9E9, 9E9, 9E9, 9E9, 9E9, 9E9]];
	VAR robtarget Openhole_1893 := [[433.54, -17.58, 181.4], [-0.056942, 0.70481, 0.705377, 0.049431], [0,0,0,0], [9E9, 9E9, 9E9, 9E9, 9E9, 9E9]];
	VAR robtarget Openhole_1894 := [[434.04, -17.59, 181.39], [-0.055259, 0.704944, 0.70549, 0.047796], [0,0,0,0], [9E9, 9E9, 9E9, 9E9, 9E9, 9E9]];
	VAR robtarget Openhole_1895 := [[434.54, -17.58, 181.39], [-0.053612, 0.705071, 0.705601, 0.046118], [0,0,0,0], [9E9, 9E9, 9E9, 9E9, 9E9, 9E9]];
	VAR robtarget Openhole_1896 := [[435.04, -17.58, 181.38], [-0.051947, 0.705196, 0.705708, 0.044453], [0,0,0,0], [9E9, 9E9, 9E9, 9E9, 9E9, 9E9]];
	VAR robtarget Openhole_1897 := [[435.54, -17.56, 181.38], [-0.050347, 0.705312, 0.705815, 0.042721], [0,0,0,0], [9E9, 9E9, 9E9, 9E9, 9E9, 9E9]];
	VAR robtarget Openhole_1898 := [[436.54, -17.57, 181.36], [-0.046982, 0.705544, 0.706008, 0.039403], [0,0,0,0], [9E9, 9E9, 9E9, 9E9, 9E9, 9E9]];
	VAR robtarget Openhole_1899 := [[437.08, -18.86, 181.2], [-0.040831, 0.705927, 0.705864, 0.041905], [0,0,0,0], [9E9, 9E9, 9E9, 9E9, 9E9, 9E9]];
	VAR robtarget Openhole_1900 := [[436.63, -19.07, 181.18], [-0.041621, 0.705881, 0.705728, 0.044138], [0,0,0,0], [9E9, 9E9, 9E9, 9E9, 9E9, 9E9]];
	VAR robtarget Openhole_1901 := [[435.69, -19.42, 181.13], [-0.043591, 0.705762, 0.705446, 0.048433], [0,0,0,0], [9E9, 9E9, 9E9, 9E9, 9E9, 9E9]];
	VAR robtarget Openhole_1902 := [[434.78, -19.82, 181.07], [-0.045288, 0.705655, 0.705131, 0.052827], [0,0,0,0], [9E9, 9E9, 9E9, 9E9, 9E9, 9E9]];
	VAR robtarget Openhole_1903 := [[434.32, -20.01, 181.04], [-0.046191, 0.705596, 0.704965, 0.054996], [0,0,0,0], [9E9, 9E9, 9E9, 9E9, 9E9, 9E9]];
	VAR robtarget Openhole_1904 := [[433.85, -20.18, 181.01], [-0.047167, 0.705532, 0.704795, 0.057129], [0,0,0,0], [9E9, 9E9, 9E9, 9E9, 9E9, 9E9]];
	VAR robtarget Openhole_1905 := [[432.42, -20.64, 180.92], [-0.050355, 0.705312, 0.704261, 0.063376], [0,0,0,0], [9E9, 9E9, 9E9, 9E9, 9E9, 9E9]];
	VAR robtarget Openhole_1906 := [[430.02, -21.29, 180.76], [-0.056167, 0.704873, 0.703285, 0.073416], [0,0,0,0], [9E9, 9E9, 9E9, 9E9, 9E9, 9E9]];
	VAR robtarget Openhole_1907 := [[429.04, -21.5, 180.7], [-0.058648, 0.70467, 0.702869, 0.077301], [0,0,0,0], [9E9, 9E9, 9E9, 9E9, 9E9, 9E9]];
	VAR robtarget Openhole_1908 := [[428.06, -21.68, 180.64], [-0.061272, 0.704447, 0.702444, 0.08107], [0,0,0,0], [9E9, 9E9, 9E9, 9E9, 9E9, 9E9]];
	VAR robtarget Openhole_1909 := [[424.09, -22.12, 180.43], [-0.072742, 0.703355, 0.700674, 0.095164], [0,0,0,0], [9E9, 9E9, 9E9, 9E9, 9E9, 9E9]];
	VAR robtarget Openhole_1910 := [[423.09, -22.18, 180.38], [-0.075744, 0.703038, 0.700212, 0.098507], [0,0,0,0], [9E9, 9E9, 9E9, 9E9, 9E9, 9E9]];
	VAR robtarget Openhole_1911 := [[418.1, -22.26, 180.21], [-0.091309, 0.701187, 0.697819, 0.114232], [0,0,0,0], [9E9, 9E9, 9E9, 9E9, 9E9, 9E9]];
	VAR robtarget Openhole_1912 := [[417.6, -22.26, 180.19], [-0.092873, 0.700981, 0.697569, 0.115749], [0,0,0,0], [9E9, 9E9, 9E9, 9E9, 9E9, 9E9]];
	VAR robtarget Openhole_1913 := [[405.6, -22.12, 179.88], [-0.129371, 0.695171, 0.690959, 0.150252], [0,0,0,0], [9E9, 9E9, 9E9, 9E9, 9E9, 9E9]];
	VAR robtarget Openhole_1914 := [[405.1, -22.12, 179.86], [-0.130807, 0.694902, 0.690655, 0.151642], [0,0,0,0], [9E9, 9E9, 9E9, 9E9, 9E9, 9E9]];
	VAR robtarget Openhole_1915 := [[397.61, -22.29, 179.56], [-0.151215, 0.690749, 0.685799, 0.172277], [0,0,0,0], [9E9, 9E9, 9E9, 9E9, 9E9, 9E9]];
	VAR robtarget Openhole_1916 := [[395.12, -22.43, 179.4], [-0.157478, 0.689348, 0.68405, 0.179098], [0,0,0,0], [9E9, 9E9, 9E9, 9E9, 9E9, 9E9]];
	VAR robtarget Openhole_1917 := [[394.34, -22.46, 179.36], [-0.159457, 0.688893, 0.683507, 0.181159], [0,0,0,0], [9E9, 9E9, 9E9, 9E9, 9E9, 9E9]];
	VAR robtarget Openhole_1918 := [[389.34, -22.46, 179.2], [-0.172368, 0.685776, 0.680121, 0.193481], [0,0,0,0], [9E9, 9E9, 9E9, 9E9, 9E9, 9E9]];
	VAR robtarget Openhole_1919 := [[362.34, -22.46, 179.28], [-0.183051, 0.683002, 0.683002, 0.183051], [0,0,0,0], [9E9, 9E9, 9E9, 9E9, 9E9, 9E9]];
	VAR robtarget Openhole_1920 := [[362.34, -23.36, 178.76], [-0.183051, 0.683002, 0.683002, 0.183051], [0,0,0,0], [9E9, 9E9, 9E9, 9E9, 9E9, 9E9]];
	VAR robtarget Openhole_1921 := [[389.34, -23.36, 178.68], [-0.169792, 0.686419, 0.679389, 0.196038], [0,0,0,0], [9E9, 9E9, 9E9, 9E9, 9E9, 9E9]];
	VAR robtarget Openhole_1922 := [[394.34, -23.36, 178.89], [-0.156817, 0.689499, 0.682806, 0.183781], [0,0,0,0], [9E9, 9E9, 9E9, 9E9, 9E9, 9E9]];
	VAR robtarget Openhole_1923 := [[395.23, -23.34, 178.94], [-0.154526, 0.690016, 0.683426, 0.181464], [0,0,0,0], [9E9, 9E9, 9E9, 9E9, 9E9, 9E9]];
	VAR robtarget Openhole_1924 := [[401.21, -23.09, 179.3], [-0.138898, 0.693331, 0.687547, 0.165166], [0,0,0,0], [9E9, 9E9, 9E9, 9E9, 9E9, 9E9]];
	VAR robtarget Openhole_1925 := [[404.71, -23.06, 179.45], [-0.129063, 0.695228, 0.689776, 0.155591], [0,0,0,0], [9E9, 9E9, 9E9, 9E9, 9E9, 9E9]];
	VAR robtarget Openhole_1926 := [[405.21, -23.06, 179.47], [-0.127621, 0.695495, 0.690085, 0.154216], [0,0,0,0], [9E9, 9E9, 9E9, 9E9, 9E9, 9E9]];
	VAR robtarget Openhole_1927 := [[417.2, -23.21, 179.89], [-0.091065, 0.701218, 0.696852, 0.119991], [0,0,0,0], [9E9, 9E9, 9E9, 9E9, 9E9, 9E9]];
	VAR robtarget Openhole_1928 := [[417.7, -23.21, 179.91], [-0.089505, 0.701419, 0.697111, 0.118477], [0,0,0,0], [9E9, 9E9, 9E9, 9E9, 9E9, 9E9]];
	VAR robtarget Openhole_1929 := [[418.2, -23.21, 179.93], [-0.087938, 0.701617, 0.697366, 0.116962], [0,0,0,0], [9E9, 9E9, 9E9, 9E9, 9E9, 9E9]];
	VAR robtarget Openhole_1930 := [[418.7, -23.21, 179.95], [-0.086379, 0.701811, 0.697622, 0.115431], [0,0,0,0], [9E9, 9E9, 9E9, 9E9, 9E9, 9E9]];
	VAR robtarget Openhole_1931 := [[423.19, -23.06, 180.17], [-0.072557, 0.703374, 0.699846, 0.101071], [0,0,0,0], [9E9, 9E9, 9E9, 9E9, 9E9, 9E9]];
	VAR robtarget Openhole_1932 := [[425.18, -22.88, 180.28], [-0.066709, 0.703953, 0.7008, 0.094229], [0,0,0,0], [9E9, 9E9, 9E9, 9E9, 9E9, 9E9]];
	VAR robtarget Openhole_1933 := [[428.14, -22.45, 180.48], [-0.058463, 0.704686, 0.702177, 0.083352], [0,0,0,0], [9E9, 9E9, 9E9, 9E9, 9E9, 9E9]];
	VAR robtarget Openhole_1934 := [[428.63, -22.36, 180.52], [-0.057173, 0.704792, 0.702399, 0.081459], [0,0,0,0], [9E9, 9E9, 9E9, 9E9, 9E9, 9E9]];
	VAR robtarget Openhole_1935 := [[430.48, -23.42, 180.38], [-0.047545, 0.705507, 0.702681, 0.078988], [0,0,0,0], [9E9, 9E9, 9E9, 9E9, 9E9, 9E9]];
	VAR robtarget Openhole_1936 := [[429.52, -23.69, 180.29], [-0.049803, 0.705351, 0.702219, 0.082995], [0,0,0,0], [9E9, 9E9, 9E9, 9E9, 9E9, 9E9]];
	VAR robtarget Openhole_1937 := [[428.07, -24.05, 180.15], [-0.053372, 0.70509, 0.701501, 0.08886], [0,0,0,0], [9E9, 9E9, 9E9, 9E9, 9E9, 9E9]];
	VAR robtarget Openhole_1938 := [[427.1, -24.27, 180.06], [-0.055857, 0.704897, 0.701007, 0.092674], [0,0,0,0], [9E9, 9E9, 9E9, 9E9, 9E9, 9E9]];
	VAR robtarget Openhole_1939 := [[426.61, -24.36, 180.01], [-0.057149, 0.704794, 0.700758, 0.094541], [0,0,0,0], [9E9, 9E9, 9E9, 9E9, 9E9, 9E9]];
	VAR robtarget Openhole_1940 := [[425.13, -24.59, 179.88], [-0.061205, 0.704453, 0.700003, 0.099976], [0,0,0,0], [9E9, 9E9, 9E9, 9E9, 9E9, 9E9]];
	VAR robtarget Openhole_1941 := [[424.15, -24.72, 179.8], [-0.064009, 0.704204, 0.699492, 0.103492], [0,0,0,0], [9E9, 9E9, 9E9, 9E9, 9E9, 9E9]];
	VAR robtarget Openhole_1942 := [[419.67, -25.03, 179.47], [-0.077376, 0.702861, 0.697134, 0.118342], [0,0,0,0], [9E9, 9E9, 9E9, 9E9, 9E9, 9E9]];
	VAR robtarget Openhole_1943 := [[416.18, -25.08, 179.25], [-0.088233, 0.70158, 0.695236, 0.129022], [0,0,0,0], [9E9, 9E9, 9E9, 9E9, 9E9, 9E9]];
	VAR robtarget Openhole_1944 := [[415.68, -25.08, 179.22], [-0.089798, 0.701382, 0.694961, 0.130498], [0,0,0,0], [9E9, 9E9, 9E9, 9E9, 9E9, 9E9]];
	VAR robtarget Openhole_1945 := [[402.2, -24.86, 178.53], [-0.130737, 0.694916, 0.686898, 0.167842], [0,0,0,0], [9E9, 9E9, 9E9, 9E9, 9E9, 9E9]];
	VAR robtarget Openhole_1946 := [[401.7, -24.86, 178.51], [-0.132152, 0.694648, 0.686571, 0.169175], [0,0,0,0], [9E9, 9E9, 9E9, 9E9, 9E9, 9E9]];
	VAR robtarget Openhole_1947 := [[395.72, -25.05, 178.08], [-0.148171, 0.691408, 0.682423, 0.185199], [0,0,0,0], [9E9, 9E9, 9E9, 9E9, 9E9, 9E9]];
	VAR robtarget Openhole_1948 := [[395.22, -25.08, 178.03], [-0.14942, 0.691139, 0.682058, 0.186538], [0,0,0,0], [9E9, 9E9, 9E9, 9E9, 9E9, 9E9]];
	VAR robtarget Openhole_1949 := [[394.34, -25.1, 177.97], [-0.151732, 0.690635, 0.681432, 0.188815], [0,0,0,0], [9E9, 9E9, 9E9, 9E9, 9E9, 9E9]];
	VAR robtarget Openhole_1950 := [[389.33, -25.1, 177.67], [-0.164832, 0.687627, 0.677953, 0.200946], [0,0,0,0], [9E9, 9E9, 9E9, 9E9, 9E9, 9E9]];
	VAR robtarget Openhole_1951 := [[362.33, -25.1, 177.76], [-0.183051, 0.683002, 0.683002, 0.183051], [0,0,0,0], [9E9, 9E9, 9E9, 9E9, 9E9, 9E9]];
	VAR robtarget Openhole_1952 := [[362.33, -25.89, 177.3], [-0.183051, 0.683002, 0.683002, 0.183051], [0,0,0,0], [9E9, 9E9, 9E9, 9E9, 9E9, 9E9]];
	VAR robtarget Openhole_1953 := [[389.33, -25.89, 177.22], [-0.162587, 0.688161, 0.677293, 0.203161], [0,0,0,0], [9E9, 9E9, 9E9, 9E9, 9E9, 9E9]];
	VAR robtarget Openhole_1954 := [[394.33, -25.89, 177.55], [-0.149431, 0.691137, 0.680798, 0.191087], [0,0,0,0], [9E9, 9E9, 9E9, 9E9, 9E9, 9E9]];
	VAR robtarget Openhole_1955 := [[395.1, -25.86, 177.61], [-0.14743, 0.691567, 0.681348, 0.189114], [0,0,0,0], [9E9, 9E9, 9E9, 9E9, 9E9, 9E9]];
	VAR robtarget Openhole_1956 := [[400.58, -25.68, 178.06], [-0.132835, 0.694518, 0.685217, 0.174578], [0,0,0,0], [9E9, 9E9, 9E9, 9E9, 9E9, 9E9]];
	VAR robtarget Openhole_1957 := [[401.58, -25.68, 178.12], [-0.130019, 0.69505, 0.685884, 0.17194], [0,0,0,0], [9E9, 9E9, 9E9, 9E9, 9E9, 9E9]];
	VAR robtarget Openhole_1958 := [[402.08, -25.68, 178.16], [-0.128595, 0.695315, 0.686213, 0.17062], [0,0,0,0], [9E9, 9E9, 9E9, 9E9, 9E9, 9E9]];
	VAR robtarget Openhole_1959 := [[416.05, -25.98, 178.95], [-0.085765, 0.701886, 0.694631, 0.13224], [0,0,0,0], [9E9, 9E9, 9E9, 9E9, 9E9, 9E9]];
	VAR robtarget Openhole_1960 := [[416.55, -25.98, 178.99], [-0.084201, 0.702076, 0.694912, 0.130757], [0,0,0,0], [9E9, 9E9, 9E9, 9E9, 9E9, 9E9]];
	VAR robtarget Openhole_1961 := [[421.53, -25.83, 179.36], [-0.068838, 0.703748, 0.69766, 0.1152], [0,0,0,0], [9E9, 9E9, 9E9, 9E9, 9E9, 9E9]];
	VAR robtarget Openhole_1962 := [[425, -25.46, 179.67], [-0.058787, 0.704659, 0.699528, 0.103248], [0,0,0,0], [9E9, 9E9, 9E9, 9E9, 9E9, 9E9]];
	VAR robtarget Openhole_1963 := [[426.96, -25.13, 179.87], [-0.053462, 0.705083, 0.700566, 0.095953], [0,0,0,0], [9E9, 9E9, 9E9, 9E9, 9E9, 9E9]];
	VAR robtarget Openhole_1964 := [[427.45, -25.03, 179.92], [-0.05221, 0.705177, 0.700823, 0.094059], [0,0,0,0], [9E9, 9E9, 9E9, 9E9, 9E9, 9E9]];
	VAR robtarget Openhole_1965 := [[430.33, -24.25, 180.23], [-0.045272, 0.705656, 0.702308, 0.082238], [0,0,0,0], [9E9, 9E9, 9E9, 9E9, 9E9, 9E9]];
	VAR robtarget Openhole_1966 := [[430.8, -24.09, 180.28], [-0.044224, 0.705722, 0.702545, 0.08019], [0,0,0,0], [9E9, 9E9, 9E9, 9E9, 9E9, 9E9]];
	VAR robtarget Openhole_1967 := [[431.73, -23.75, 180.38], [-0.042273, 0.705842, 0.70301, 0.076008], [0,0,0,0], [9E9, 9E9, 9E9, 9E9, 9E9, 9E9]];
	VAR robtarget Openhole_1968 := [[432.19, -23.56, 180.43], [-0.041356, 0.705896, 0.703236, 0.073883], [0,0,0,0], [9E9, 9E9, 9E9, 9E9, 9E9, 9E9]];
	VAR robtarget Openhole_1969 := [[432.65, -23.37, 180.48], [-0.040478, 0.705947, 0.703458, 0.071738], [0,0,0,0], [9E9, 9E9, 9E9, 9E9, 9E9, 9E9]];
	VAR robtarget Openhole_1970 := [[433.55, -22.94, 180.59], [-0.03889, 0.706037, 0.70389, 0.067368], [0,0,0,0], [9E9, 9E9, 9E9, 9E9, 9E9, 9E9]];
	VAR robtarget Openhole_1971 := [[434, -22.72, 180.64], [-0.038158, 0.706076, 0.704099, 0.065156], [0,0,0,0], [9E9, 9E9, 9E9, 9E9, 9E9, 9E9]];
	VAR robtarget Openhole_1972 := [[434.43, -22.48, 180.69], [-0.037487, 0.706112, 0.704302, 0.062919], [0,0,0,0], [9E9, 9E9, 9E9, 9E9, 9E9, 9E9]];
	VAR robtarget Openhole_1973 := [[435.29, -21.98, 180.78], [-0.03628, 0.706175, 0.704692, 0.058394], [0,0,0,0], [9E9, 9E9, 9E9, 9E9, 9E9, 9E9]];
	VAR robtarget Openhole_1974 := [[435.72, -21.72, 180.83], [-0.035738, 0.706203, 0.704877, 0.05611], [0,0,0,0], [9E9, 9E9, 9E9, 9E9, 9E9, 9E9]];
	VAR robtarget Openhole_1975 := [[436.14, -21.45, 180.87], [-0.035238, 0.706228, 0.705056, 0.053811], [0,0,0,0], [9E9, 9E9, 9E9, 9E9, 9E9, 9E9]];
	VAR robtarget Openhole_1976 := [[436.96, -20.89, 180.96], [-0.034375, 0.706271, 0.705395, 0.049176], [0,0,0,0], [9E9, 9E9, 9E9, 9E9, 9E9, 9E9]];
	VAR robtarget Openhole_1977 := [[437.76, -20.3, 181.04], [-0.033682, 0.706304, 0.705705, 0.044497], [0,0,0,0], [9E9, 9E9, 9E9, 9E9, 9E9, 9E9]];
	VAR robtarget Openhole_1978 := [[438.17, -20.01, 181.08], [-0.033275, 0.706323, 0.705849, 0.042161], [0,0,0,0], [9E9, 9E9, 9E9, 9E9, 9E9, 9E9]];
	VAR robtarget Openhole_1979 := [[441.8, -21.35, 181.01], [-0.016492, 0.706914, 0.706266, 0.034481], [0,0,0,0], [9E9, 9E9, 9E9, 9E9, 9E9, 9E9]];
	VAR robtarget Openhole_1980 := [[441.01, -21.74, 180.96], [-0.017844, 0.706882, 0.70606, 0.038469], [0,0,0,0], [9E9, 9E9, 9E9, 9E9, 9E9, 9E9]];
	VAR robtarget Openhole_1981 := [[440.59, -22.01, 180.93], [-0.018352, 0.706869, 0.705929, 0.040795], [0,0,0,0], [9E9, 9E9, 9E9, 9E9, 9E9, 9E9]];
	VAR robtarget Openhole_1982 := [[439.34, -22.84, 180.81], [-0.019766, 0.70683, 0.705491, 0.047776], [0,0,0,0], [9E9, 9E9, 9E9, 9E9, 9E9, 9E9]];
	VAR robtarget Openhole_1983 := [[438.06, -23.61, 180.68], [-0.021475, 0.706781, 0.704991, 0.054658], [0,0,0,0], [9E9, 9E9, 9E9, 9E9, 9E9, 9E9]];
	VAR robtarget Openhole_1984 := [[437.63, -23.85, 180.64], [-0.022149, 0.70676, 0.704812, 0.056917], [0,0,0,0], [9E9, 9E9, 9E9, 9E9, 9E9, 9E9]];
	VAR robtarget Openhole_1985 := [[435.85, -24.75, 180.44], [-0.025112, 0.706661, 0.704036, 0.065827], [0,0,0,0], [9E9, 9E9, 9E9, 9E9, 9E9, 9E9]];
	VAR robtarget Openhole_1986 := [[432.92, -27.42, 179.86], [-0.02603, 0.706628, 0.702061, 0.084324], [0,0,0,0], [9E9, 9E9, 9E9, 9E9, 9E9, 9E9]];
	VAR robtarget Openhole_1987 := [[434.35, -26.98, 180.03], [-0.022691, 0.706743, 0.702766, 0.078229], [0,0,0,0], [9E9, 9E9, 9E9, 9E9, 9E9, 9E9]];
	VAR robtarget Openhole_1988 := [[438.55, -25.44, 180.51], [-0.013667, 0.706975, 0.704624, 0.059203], [0,0,0,0], [9E9, 9E9, 9E9, 9E9, 9E9, 9E9]];
	VAR robtarget Openhole_1989 := [[439.46, -25.04, 180.61], [-0.011931, 0.707006, 0.704979, 0.054813], [0,0,0,0], [9E9, 9E9, 9E9, 9E9, 9E9, 9E9]];
	VAR robtarget Openhole_1990 := [[439.91, -24.83, 180.65], [-0.01111, 0.70702, 0.705148, 0.052594], [0,0,0,0], [9E9, 9E9, 9E9, 9E9, 9E9, 9E9]];
	VAR robtarget Openhole_1991 := [[440.8, -24.39, 180.74], [-0.009577, 0.707042, 0.705468, 0.048109], [0,0,0,0], [9E9, 9E9, 9E9, 9E9, 9E9, 9E9]];
	VAR robtarget Openhole_1992 := [[441.23, -24.14, 180.78], [-0.008965, 0.70705, 0.705621, 0.045816], [0,0,0,0], [9E9, 9E9, 9E9, 9E9, 9E9, 9E9]];
	VAR robtarget Openhole_1993 := [[441.65, -23.86, 180.82], [-0.008478, 0.707056, 0.705768, 0.043489], [0,0,0,0], [9E9, 9E9, 9E9, 9E9, 9E9, 9E9]];
	VAR robtarget Openhole_1994 := [[442.05, -23.57, 180.86], [-0.008094, 0.70706, 0.705909, 0.041141], [0,0,0,0], [9E9, 9E9, 9E9, 9E9, 9E9, 9E9]];
	VAR robtarget Openhole_1995 := [[442.67, -23.11, 180.92], [-0.007566, 0.707066, 0.706112, 0.037497], [0,0,0,0], [9E9, 9E9, 9E9, 9E9, 9E9, 9E9]];
	VAR robtarget Openhole_1996 := [[445.06, -25.46, 180.92], [0.008532, 0.707055, 0.706119, 0.037358], [0,0,0,0], [9E9, 9E9, 9E9, 9E9, 9E9, 9E9]];
	VAR robtarget Openhole_1997 := [[444.45, -25.91, 180.86], [0.008002, 0.707062, 0.70592, 0.040959], [0,0,0,0], [9E9, 9E9, 9E9, 9E9, 9E9, 9E9]];
	VAR robtarget Openhole_1998 := [[443.53, -26.29, 180.77], [0.006153, 0.70708, 0.705651, 0.045354], [0,0,0,0], [9E9, 9E9, 9E9, 9E9, 9E9, 9E9]];
	VAR robtarget Openhole_1999 := [[443.06, -26.45, 180.73], [0.005072, 0.707089, 0.705511, 0.047475], [0,0,0,0], [9E9, 9E9, 9E9, 9E9, 9E9, 9E9]];
	VAR robtarget Openhole_2000 := [[442.1, -26.73, 180.64], [0.002759, 0.707101, 0.705219, 0.051632], [0,0,0,0], [9E9, 9E9, 9E9, 9E9, 9E9, 9E9]];
	VAR robtarget Openhole_2001 := [[441.62, -26.84, 180.6], [0.001469, 0.707105, 0.70507, 0.053629], [0,0,0,0], [9E9, 9E9, 9E9, 9E9, 9E9, 9E9]];
	VAR robtarget Openhole_2002 := [[437.75, -27.77, 180.21], [-0.008531, 0.707055, 0.703666, 0.069668], [0,0,0,0], [9E9, 9E9, 9E9, 9E9, 9E9, 9E9]];
	VAR robtarget Openhole_2003 := [[431.47, -29.27, 179.42], [-0.024733, 0.706674, 0.700677, 0.095137], [0,0,0,0], [9E9, 9E9, 9E9, 9E9, 9E9, 9E9]];
	VAR robtarget Openhole_2004 := [[428.05, -31.34, 178.66], [-0.029362, 0.706497, 0.698054, 0.112787], [0,0,0,0], [9E9, 9E9, 9E9, 9E9, 9E9, 9E9]];
	VAR robtarget Openhole_2005 := [[437.85, -29.84, 179.99], [-0.001274, 0.707106, 0.702987, 0.07622], [0,0,0,0], [9E9, 9E9, 9E9, 9E9, 9E9, 9E9]];
	VAR robtarget Openhole_2006 := [[439.82, -29.61, 180.21], [0.004659, 0.707091, 0.703742, 0.068902], [0,0,0,0], [9E9, 9E9, 9E9, 9E9, 9E9, 9E9]];
	VAR robtarget Openhole_2007 := [[441.81, -29.49, 180.42], [0.011031, 0.707021, 0.704393, 0.061886], [0,0,0,0], [9E9, 9E9, 9E9, 9E9, 9E9, 9E9]];
	VAR robtarget Openhole_2008 := [[443.3, -29.47, 180.57], [0.016041, 0.706925, 0.704821, 0.056806], [0,0,0,0], [9E9, 9E9, 9E9, 9E9, 9E9, 9E9]];
	VAR robtarget Openhole_2009 := [[450.76, -29.75, 181.33], [0.042348, 0.705838, 0.706359, 0.032507], [0,0,0,0], [9E9, 9E9, 9E9, 9E9, 9E9, 9E9]];
	VAR robtarget Openhole_2010 := [[451.25, -29.75, 181.38], [0.044036, 0.705734, 0.706435, 0.030816], [0,0,0,0], [9E9, 9E9, 9E9, 9E9, 9E9, 9E9]];
	VAR robtarget Openhole_2011 := [[451.75, -29.75, 181.43], [0.045708, 0.705628, 0.706507, 0.029111], [0,0,0,0], [9E9, 9E9, 9E9, 9E9, 9E9, 9E9]];
	VAR robtarget Openhole_2012 := [[455.72, -29.42, 181.82], [0.05799, 0.704725, 0.706958, 0.014496], [0,0,0,0], [9E9, 9E9, 9E9, 9E9, 9E9, 9E9]];
	VAR robtarget Openhole_2013 := [[458.68, -29.06, 182.08], [0.066673, 0.703956, 0.7071, 0.003149], [0,0,0,0], [9E9, 9E9, 9E9, 9E9, 9E9, 9E9]];
	VAR robtarget Openhole_2014 := [[468.12, -28.35, 182.87], [0.095173, 0.700673, 0.706419, -0.031187], [0,0,0,0], [9E9, 9E9, 9E9, 9E9, 9E9, 9E9]];
	VAR robtarget Openhole_2015 := [[481.57, -27.6, 183.84], [0.134313, 0.694233, 0.702841, -0.077557], [0,0,0,0], [9E9, 9E9, 9E9, 9E9, 9E9, 9E9]];
	VAR robtarget Openhole_2016 := [[483.56, -27.51, 183.98], [0.139902, 0.693129, 0.702085, -0.084122], [0,0,0,0], [9E9, 9E9, 9E9, 9E9, 9E9, 9E9]];
	VAR robtarget Openhole_2017 := [[481.54, -17.51, 180.71], [0.102006, 0.699711, 0.6985, -0.10999], [0,0,0,0], [9E9, 9E9, 9E9, 9E9, 9E9, 9E9]];
	VAR robtarget Openhole_2018 := [[491.04, -17.63, 180.62], [0.13071, 0.694921, 0.69355, -0.137801], [0,0,0,0], [9E9, 9E9, 9E9, 9E9, 9E9, 9E9]];
	VAR robtarget Openhole_2019 := [[491.54, -17.62, 180.61], [0.132146, 0.694649, 0.693263, -0.139235], [0,0,0,0], [9E9, 9E9, 9E9, 9E9, 9E9, 9E9]];
	VAR robtarget Openhole_2020 := [[500.54, -17.43, 180.4], [0.156537, 0.689562, 0.687678, -0.164616], [0,0,0,0], [9E9, 9E9, 9E9, 9E9, 9E9, 9E9]];
	VAR robtarget Openhole_2021 := [[503.53, -17.27, 180.27], [0.163979, 0.687831, 0.685636, -0.172925], [0,0,0,0], [9E9, 9E9, 9E9, 9E9, 9E9, 9E9]];
	VAR robtarget Openhole_2022 := [[504.34, -17.24, 180.24], [0.166003, 0.687345, 0.685082, -0.175106], [0,0,0,0], [9E9, 9E9, 9E9, 9E9, 9E9, 9E9]];
	VAR robtarget Openhole_2023 := [[509.34, -17.24, 180.15], [0.183051, 0.683002, 0.683002, -0.183051], [0,0,0,0], [9E9, 9E9, 9E9, 9E9, 9E9, 9E9]];
	VAR robtarget Openhole_2024 := [[536.34, -17.24, 180.06], [0.183051, 0.683002, 0.683002, -0.183051], [0,0,0,0], [9E9, 9E9, 9E9, 9E9, 9E9, 9E9]];
	VAR robtarget Openhole_2025 := [[536.34, -17.96, 180.48], [0.183051, 0.683002, 0.683002, -0.183051], [0,0,0,0], [9E9, 9E9, 9E9, 9E9, 9E9, 9E9]];
	VAR robtarget Openhole_2026 := [[509.34, -17.96, 180.57], [0.183051, 0.683002, 0.683002, -0.183051], [0,0,0,0], [9E9, 9E9, 9E9, 9E9, 9E9, 9E9]];
	VAR robtarget Openhole_2027 := [[504.34, -17.96, 180.62], [0.168111, 0.686832, 0.685617, -0.173002], [0,0,0,0], [9E9, 9E9, 9E9, 9E9, 9E9, 9E9]];
	VAR robtarget Openhole_2028 := [[496.08, -18.29, 180.85], [0.146993, 0.69166, 0.691022, -0.149962], [0,0,0,0], [9E9, 9E9, 9E9, 9E9, 9E9, 9E9]];
	VAR robtarget Openhole_2029 := [[491.08, -18.34, 180.91], [0.13304, 0.694478, 0.693963, -0.135705], [0,0,0,0], [9E9, 9E9, 9E9, 9E9, 9E9, 9E9]];
	VAR robtarget Openhole_2030 := [[490.58, -18.34, 180.91], [0.1316, 0.694753, 0.694243, -0.134264], [0,0,0,0], [9E9, 9E9, 9E9, 9E9, 9E9, 9E9]];
	VAR robtarget Openhole_2031 := [[474.59, -18.11, 180.96], [0.082163, 0.702317, 0.701826, -0.086259], [0,0,0,0], [9E9, 9E9, 9E9, 9E9, 9E9, 9E9]];
	VAR robtarget Openhole_2032 := [[474.09, -18.11, 180.96], [0.080569, 0.702502, 0.702021, -0.084658], [0,0,0,0], [9E9, 9E9, 9E9, 9E9, 9E9, 9E9]];
	VAR robtarget Openhole_2033 := [[471.09, -18.16, 181], [0.07107, 0.703526, 0.703135, -0.074839], [0,0,0,0], [9E9, 9E9, 9E9, 9E9, 9E9, 9E9]];
	VAR robtarget Openhole_2034 := [[469.59, -18.24, 181.03], [0.066457, 0.703977, 0.703662, -0.069709], [0,0,0,0], [9E9, 9E9, 9E9, 9E9, 9E9, 9E9]];
	VAR robtarget Openhole_2035 := [[467.1, -18.42, 181.08], [0.05889, 0.70465, 0.704477, -0.060928], [0,0,0,0], [9E9, 9E9, 9E9, 9E9, 9E9, 9E9]];
	VAR robtarget Openhole_2036 := [[466.6, -18.47, 181.09], [0.057444, 0.70477, 0.704633, -0.059098], [0,0,0,0], [9E9, 9E9, 9E9, 9E9, 9E9, 9E9]];
	VAR robtarget Openhole_2037 := [[467.28, -16.77, 180.79], [0.053993, 0.705042, 0.703921, -0.067043], [0,0,0,0], [9E9, 9E9, 9E9, 9E9, 9E9, 9E9]];
	VAR robtarget Openhole_2038 := [[468.25, -16.53, 180.73], [0.056398, 0.704854, 0.703532, -0.07101], [0,0,0,0], [9E9, 9E9, 9E9, 9E9, 9E9, 9E9]];
	VAR robtarget Openhole_2039 := [[469.23, -16.32, 180.66], [0.058893, 0.70465, 0.703129, -0.074899], [0,0,0,0], [9E9, 9E9, 9E9, 9E9, 9E9, 9E9]];
	VAR robtarget Openhole_2040 := [[469.71, -16.22, 180.63], [0.060178, 0.704541, 0.702923, -0.076811], [0,0,0,0], [9E9, 9E9, 9E9, 9E9, 9E9, 9E9]];
	VAR robtarget Openhole_2041 := [[470.21, -16.14, 180.6], [0.061499, 0.704427, 0.702714, -0.078692], [0,0,0,0], [9E9, 9E9, 9E9, 9E9, 9E9, 9E9]];
	VAR robtarget Openhole_2042 := [[472.19, -15.88, 180.49], [0.067086, 0.703917, 0.701866, -0.085935], [0,0,0,0], [9E9, 9E9, 9E9, 9E9, 9E9, 9E9]];
	VAR robtarget Openhole_2043 := [[473.18, -15.79, 180.44], [0.070019, 0.703632, 0.701432, -0.089407], [0,0,0,0], [9E9, 9E9, 9E9, 9E9, 9E9, 9E9]];
	VAR robtarget Openhole_2044 := [[478.67, -15.58, 180.21], [0.086859, 0.701752, 0.698911, -0.107347], [0,0,0,0], [9E9, 9E9, 9E9, 9E9, 9E9, 9E9]];
	VAR robtarget Openhole_2045 := [[479.17, -15.58, 180.19], [0.088427, 0.701556, 0.698672, -0.108894], [0,0,0,0], [9E9, 9E9, 9E9, 9E9, 9E9, 9E9]];
	VAR robtarget Openhole_2046 := [[479.67, -15.58, 180.18], [0.089994, 0.701357, 0.69843, -0.110433], [0,0,0,0], [9E9, 9E9, 9E9, 9E9, 9E9, 9E9]];
	VAR robtarget Openhole_2047 := [[492.66, -15.73, 179.81], [0.129524, 0.695143, 0.691391, -0.148252], [0,0,0,0], [9E9, 9E9, 9E9, 9E9, 9E9, 9E9]];
	VAR robtarget Openhole_2048 := [[493.16, -15.73, 179.79], [0.130954, 0.694875, 0.691088, -0.149657], [0,0,0,0], [9E9, 9E9, 9E9, 9E9, 9E9, 9E9]];
	VAR robtarget Openhole_2049 := [[500.65, -15.57, 179.47], [0.151314, 0.690727, 0.686255, -0.170454], [0,0,0,0], [9E9, 9E9, 9E9, 9E9, 9E9, 9E9]];
	VAR robtarget Openhole_2050 := [[503.64, -15.39, 179.28], [0.158756, 0.689055, 0.684148, -0.17872], [0,0,0,0], [9E9, 9E9, 9E9, 9E9, 9E9, 9E9]];
	VAR robtarget Openhole_2051 := [[504.34, -15.36, 179.24], [0.160495, 0.688652, 0.683658, -0.180586], [0,0,0,0], [9E9, 9E9, 9E9, 9E9, 9E9, 9E9]];
	VAR robtarget Openhole_2052 := [[509.34, -15.36, 179.06], [0.183051, 0.683002, 0.683002, -0.183051], [0,0,0,0], [9E9, 9E9, 9E9, 9E9, 9E9, 9E9]];
	VAR robtarget Openhole_2053 := [[536.34, -15.36, 178.98], [0.183051, 0.683002, 0.683002, -0.183051], [0,0,0,0], [9E9, 9E9, 9E9, 9E9, 9E9, 9E9]];
	VAR robtarget Openhole_2054 := [[536.34, -14.15, 178.28], [0.183051, 0.683002, 0.683002, -0.183051], [0,0,0,0], [9E9, 9E9, 9E9, 9E9, 9E9, 9E9]];
	VAR robtarget Openhole_2055 := [[509.34, -14.15, 178.36], [0.183051, 0.683002, 0.683002, -0.183051], [0,0,0,0], [9E9, 9E9, 9E9, 9E9, 9E9, 9E9]];
	VAR robtarget Openhole_2056 := [[504.34, -14.15, 178.6], [0.156958, 0.689467, 0.682722, -0.184093], [0,0,0,0], [9E9, 9E9, 9E9, 9E9, 9E9, 9E9]];
	VAR robtarget Openhole_2057 := [[498.3, -14.46, 179.03], [0.141545, 0.692795, 0.686978, -0.167515], [0,0,0,0], [9E9, 9E9, 9E9, 9E9, 9E9, 9E9]];
	VAR robtarget Openhole_2058 := [[493.8, -14.52, 179.25], [0.129056, 0.69523, 0.689878, -0.15514], [0,0,0,0], [9E9, 9E9, 9E9, 9E9, 9E9, 9E9]];
	VAR robtarget Openhole_2059 := [[493.3, -14.52, 179.27], [0.12762, 0.695495, 0.690188, -0.153757], [0,0,0,0], [9E9, 9E9, 9E9, 9E9, 9E9, 9E9]];
	VAR robtarget Openhole_2060 := [[480.81, -14.37, 179.77], [0.089662, 0.701399, 0.697222, -0.11782], [0,0,0,0], [9E9, 9E9, 9E9, 9E9, 9E9, 9E9]];
	VAR robtarget Openhole_2061 := [[480.31, -14.37, 179.79], [0.088108, 0.701596, 0.697479, -0.116291], [0,0,0,0], [9E9, 9E9, 9E9, 9E9, 9E9, 9E9]];
	VAR robtarget Openhole_2062 := [[475.32, -14.53, 180.06], [0.072779, 0.703351, 0.699953, -0.100331], [0,0,0,0], [9E9, 9E9, 9E9, 9E9, 9E9, 9E9]];
	VAR robtarget Openhole_2063 := [[472.34, -14.82, 180.25], [0.064116, 0.704194, 0.701366, -0.089923], [0,0,0,0], [9E9, 9E9, 9E9, 9E9, 9E9, 9E9]];
	VAR robtarget Openhole_2064 := [[471.85, -14.89, 180.29], [0.062743, 0.704318, 0.701596, -0.08811], [0,0,0,0], [9E9, 9E9, 9E9, 9E9, 9E9, 9E9]];
	VAR robtarget Openhole_2065 := [[471.36, -14.97, 180.32], [0.061405, 0.704436, 0.701825, -0.086264], [0,0,0,0], [9E9, 9E9, 9E9, 9E9, 9E9, 9E9]];
	VAR robtarget Openhole_2066 := [[469.41, -15.37, 180.48], [0.056335, 0.704859, 0.702721, -0.078631], [0,0,0,0], [9E9, 9E9, 9E9, 9E9, 9E9, 9E9]];
	VAR robtarget Openhole_2067 := [[468.44, -15.62, 180.56], [0.053996, 0.705042, 0.703154, -0.074659], [0,0,0,0], [9E9, 9E9, 9E9, 9E9, 9E9, 9E9]];
	VAR robtarget Openhole_2068 := [[467.01, -16.05, 180.68], [0.050687, 0.705288, 0.703776, -0.068548], [0,0,0,0], [9E9, 9E9, 9E9, 9E9, 9E9, 9E9]];
	VAR robtarget Openhole_2069 := [[466.54, -16.21, 180.72], [0.049686, 0.705359, 0.703978, -0.06645], [0,0,0,0], [9E9, 9E9, 9E9, 9E9, 9E9, 9E9]];
	VAR robtarget Openhole_2070 := [[465.61, -16.58, 180.8], [0.047819, 0.705488, 0.704368, -0.062177], [0,0,0,0], [9E9, 9E9, 9E9, 9E9, 9E9, 9E9]];
	VAR robtarget Openhole_2071 := [[465.15, -16.77, 180.84], [0.046929, 0.705548, 0.704555, -0.060015], [0,0,0,0], [9E9, 9E9, 9E9, 9E9, 9E9, 9E9]];
	VAR robtarget Openhole_2072 := [[463.78, -17.37, 180.95], [0.044421, 0.70571, 0.705085, -0.053439], [0,0,0,0], [9E9, 9E9, 9E9, 9E9, 9E9, 9E9]];
	VAR robtarget Openhole_2073 := [[462.86, -17.76, 181.02], [0.042658, 0.705819, 0.705402, -0.049068], [0,0,0,0], [9E9, 9E9, 9E9, 9E9, 9E9, 9E9]];
	VAR robtarget Openhole_2074 := [[462.42, -18, 181.05], [0.041978, 0.70586, 0.705556, -0.046806], [0,0,0,0], [9E9, 9E9, 9E9, 9E9, 9E9, 9E9]];
